// TwinCAT 3 PLC project SpeedControl
// ProgramVersion: 3.1.4020.4
// libraries:
//   Tc2_Drive, * (Beckhoff Automation GmbH)
//   Tc2_EtherCAT, * (Beckhoff Automation GmbH)
//   Tc2_MC2, * (Beckhoff Automation GmbH)
//   Tc2_Standard, * (Beckhoff Automation GmbH)
//   Tc2_System, * (Beckhoff Automation GmbH)
//   Tc2_Utilities, * (Beckhoff Automation GmbH)
//   Tc3_Module, * (Beckhoff Automation GmbH)
// project tree:
//   DUTs/ ST_COM_FTL_SpdCntrl.TcDUT, ST_COM_SpdCntrl_FTL.TcDUT, ST_COM_SpeedControl_IMD.TcDUT, ST_COM_IMD_SpdCntrl.TcDUT, ST_COM_SpeedControl_FTL.TcDUT, ST_MachPar.TcDUT, ST_OEE.TcDUT, ST_PowerMeasurement.TcDUT, ST_ProdPar.TcDUT, ST_ProductPar.TcDUT, ST_COM_SpdCntrl_IMD.TcDUT, ST_SysPar.TcDUT
//   GVLs/ GVL.TcGVL
//   / PlcTask_SpeedControl.TcTTO, RecipeManager.TcRMO (not stored)
//   POUs/SpeedControl/ FB_BlowOff.TcPOU, ST_BlowOffMachPar.TcDUT, ST_BlowOffErrors.TcDUT, ST_BlowOffProdPar.TcDUT, FB_Conveyor.TcPOU, ST_ConveyorErrors.TcDUT, ST_ConveyorMachPar.TcDUT, ST_ConveyorProdPar.TcDUT, ST_ConveyorSysPar.TcDUT
//   POUs/ HMI.TcPOU, MAIN.TcPOU, ST_Errors.TcDUT
//   Standard/ FB_Blink.TcPOU, FB_EthercatDiag.TcPOU
//   Standard/Motor/ FB_Motor.TcPOU, FB_MotorSS.TcPOU, ST_MotorErrors.TcDUT, ST_MotorSSErrors.TcDUT
//   Standard/NC_Axis/ FB_NcAxis.TcPOU, ST_NcAxis_Errors.TcDUT, ST_NcAxis_Parameters_XX.TcDUT, ST_NcAxis_SysPar.TcDUT
// (motion and I/O tree: see PLC project imd_plc)
// real-time tasks:
//   TASK PlcTask: cycle T#10ms, priority 20, ADS port 350
//   TASK PlcTask_SpeedControl: cycle T#2ms, priority 19, ADS port 351
// variable links:
//   IMD_PLC/IMD_PLC Instance <-> SpeedControl/SpeedControl Instance
//     PlcTask Inputs/MAIN.ComSC.SpeedControl_IMD <-> PlcTask_SpeedControl Outputs/MAIN.ComSpeedControl_IMD1.SpeedControl_IMD
//     PlcTask Outputs/MAIN.ComSC.IMD_SpeedControl <-> PlcTask_SpeedControl Inputs/MAIN.ComSpeedControl_IMD1.IMD_SpeedControl
//   SpeedControl/SpeedControl Instance <-> Device 2 (EtherCAT)/MCC01_2_610A1 (EK1100)/610A2 (EK1122)/Drive A-Belt / B-Spraybar (AX5201-0000-0203)
//     PlcTask_SpeedControl Inputs/MAIN.Conveyor.Belt.iDriveRef/aNetId <-> InfoData/AdsAddr/netId
//     PlcTask_SpeedControl Inputs/MAIN.Conveyor.Belt.iDriveRef/nDriveNo <-> InfoData/Chn0
//     PlcTask_SpeedControl Inputs/MAIN.Conveyor.Belt.iDriveRef/nSlaveAddr <-> InfoData/AdsAddr/port
//   SpeedControl/SpeedControl Instance <-> Device 2 (EtherCAT)/MCC01_2_610A1 (EK1100)/610A2 (EK1122)/EJBox (EP9128-0021)/EPP_SensorSpeedControl (EPP1322-0001)/Box SpeedControl (EPP6228-0022)
//     PlcTask_SpeedControl Inputs/MAIN.Conveyor.IMD1_GantryB.miSensorPitchClear <-> Module 11 (Digital Inputs)/Digital Inputs/Pin2 Ch1
//   SpeedControl/SpeedControl Instance <-> NC-Task 1 SAF/Axes/Conveyor
//     PlcTask_SpeedControl Inputs/MAIN.Conveyor.Belt.axAxis.NcToPlc <-> Outputs/ToPlc
//     PlcTask_SpeedControl Outputs/MAIN.Conveyor.Belt.axAxis.PlcToNc <-> Inputs/FromPlc

CONFIGURATION SpeedControl
    RESOURCE PLC ON TwinCAT3
        TASK PlcTask_SpeedControl(INTERVAL := T#2ms, PRIORITY := 19);
        PROGRAM MAIN WITH PlcTask_SpeedControl : MAIN;
    END_RESOURCE
END_CONFIGURATION

// ---- DUTs/ST_COM_FTL_SpdCntrl.TcDUT
TYPE ST_COM_FTL_SpdCntrl :
STRUCT
	MaximumSpeed	: LREAL; //(KO, amount of sheets/min)
	RTO				: BOOL;	//FTL is Ready to Operate state
	Stop			: BOOL;
	ES				: BOOL;
END_STRUCT
END_TYPE

// ---- DUTs/ST_COM_SpdCntrl_FTL.TcDUT
TYPE ST_COM_SpdCntrl_FTL :
STRUCT
	ReadyToRun			: BOOL;
	ES					: BOOL;
END_STRUCT
END_TYPE

// ---- DUTs/ST_COM_SpeedControl_IMD.TcDUT
TYPE ST_COM_SpeedControl_IMD :
STRUCT
	//Speedcontrol - IMD
	IMD_SpeedControl		AT %I* :ST_COM_IMD_SpdCntrl;
	SpeedControl_IMD		AT %Q* :ST_COM_SpdCntrl_IMD;
END_STRUCT
END_TYPE

// ---- DUTs/ST_COM_IMD_SpdCntrl.TcDUT
TYPE ST_COM_IMD_SpdCntrl :
STRUCT
	Stopped				: BOOL;					// IMD is in stopped state
	RTO					: BOOL;					// IMD is Ready to Operate state
	BlowOffProcessedA	: ARRAY[1..4] OF BOOL;	// signal to confirm that the blowoff has actually happend for A side
	BlowOffProcessedB	: ARRAY[1..4] OF BOOL;	// signal to confirm that the blowoff has actually happend for B side
	FormingReadyA		: BOOL;					// signal to confirm that the forming has actually started for A side
	FormingReadyB		: BOOL;					// signal to confirm that the forming has actually started for B side
	GantryA_Ready		: BOOL; 				// signal that Gantry A is in position above the conveyor and ready to blow off
	GantryB_Ready		: BOOL; 				// signal that Gantry B is in position above the conveyor and ready to blow off
	ES					: BOOL;					// Emergency stop from the IMD that also need to stop the conveyor
	MaximumSpeed		: REAL;					// theoretical maximum speed with current settings
	ActualSpeed			: REAL;					// Number of KO's in last cycle
	HMI_Reset			: BOOL;					// MZE 20190311 For testing at LoodsLanghout
END_STRUCT
END_TYPE

// ---- DUTs/ST_COM_SpeedControl_FTL.TcDUT
TYPE ST_COM_SpeedControl_FTL :
STRUCT
	//Speedcontrol - FTL
	FTL_SpeedControl		AT %I* :ST_COM_FTL_SpdCntrl;
	SpeedControl_FTL		AT %Q* :ST_COM_SpdCntrl_FTL;
END_STRUCT
END_TYPE

// ---- DUTs/ST_MachPar.TcDUT
TYPE ST_MachPar :
STRUCT
	Conveyor				: ST_ConveyorMachPar;
END_STRUCT
END_TYPE

// ---- DUTs/ST_OEE.TcDUT
TYPE ST_OEE :
STRUCT
	AmountOfSheets			 		: DINT;
	AmoundOfProductsSheets			: DINT;
	
END_STRUCT
END_TYPE

// ---- DUTs/ST_PowerMeasurement.TcDUT
TYPE ST_PowerMeasurement :
STRUCT
	ixPDOToggle		:BOOL;
	iwCurrent 		:DINT;
	iwVoltage		:DINT;
	iwActivePower	:DINT;
	iwIndex			:USINT;
	iwVariantValue	:DINT;
END_STRUCT
END_TYPE

// ---- DUTs/ST_ProdPar.TcDUT
TYPE ST_ProdPar :
STRUCT
	Conveyor			: ST_ConveyorProdPar;
	Product				: ST_ProductPar;
END_STRUCT
END_TYPE

// ---- DUTs/ST_ProductPar.TcDUT
TYPE ST_ProductPar :
STRUCT
	PlaceHolder			: BOOL;
END_STRUCT
END_TYPE

// ---- DUTs/ST_COM_SpdCntrl_IMD.TcDUT
TYPE ST_COM_SpdCntrl_IMD :
STRUCT
	StartFormingA		: BOOL;	//Speedcontrol needs the IMD to start froming for A side	
	StartFormingB		: BOOL;	//Speedcontrol needs the IMD to start froming for B side	
	StopForming			: BOOL;	//Speedcontrol needs the IMD to stop forming 
	BlowOffPulseA		: ARRAY[1..4] OF BOOL; 	//Blowoff pulses for A side
	BlowOffPulseB		: ARRAY[1..4] OF BOOL;	//Blowoff pulses for B side
	ErrSlotANotFree		: BOOL;					//Current slot for gantry A blow off was not free
	ErrSlotBNotFree		: BOOL;					//Current slot for gantry B blow off was not free	
	Modulo				: LREAL;				//Actual modulo position of the belt  
	SpeedInKo			: LREAL;				//Actual Speed that speedcontrol is dictating to the IMD
	PocketA_Blocked		: BOOL;					//Pocket is occupied and gantry is not allowed to blow off
	PocketB_Blocked		: BOOL;					//Pocket is occupied and gantry is not allowed to blow off
	ProdParameters		: ST_BlowOffProdPar;
END_STRUCT
END_TYPE

// ---- DUTs/ST_SysPar.TcDUT
TYPE ST_SysPar :
STRUCT
	Conveyor					: ST_ConveyorSysPar;
END_STRUCT
END_TYPE

// ---- POUs/SpeedControl/ST_BlowOffMachPar.TcDUT
TYPE ST_BlowOffMachPar :
STRUCT
	NrOfPitchMissedAlarm		: DINT;
END_STRUCT
END_TYPE

// ---- POUs/SpeedControl/ST_BlowOffErrors.TcDUT
TYPE ST_BlowOffErrors :
STRUCT
	PitchNotFree_Error		: BOOL;	//Designated pitch for blow off not free	
END_STRUCT
END_TYPE

// ---- POUs/SpeedControl/ST_BlowOffProdPar.TcDUT
TYPE ST_BlowOffProdPar :
STRUCT
	PitchGantry					: DINT;	//Pitch distance between sheets on gantry
	NrOfSheets					: DINT;	//Amount of sheets used on IMD
	NrOfCavities				: DINT;  // The amount of cavities (products) in one sheet.
	Modulo						: LREAL; //System parameter (5180)
	ModuloOffsetSensorFree		: REAL; //Offset on the modulo to start measuring if the pitch is free for dropping
	ModuloDetectionSensorFree	: REAL;	//How long the sensor needs to be active before alarm/skipping blow off based on modulo length
	SheetSize					: REAL;	//The width of a sheet
END_STRUCT
END_TYPE

// ---- POUs/SpeedControl/ST_ConveyorErrors.TcDUT
TYPE ST_ConveyorErrors :
STRUCT
	NCAxisError					: ST_NcAxis_Errors;
	
END_STRUCT
END_TYPE

// ---- POUs/SpeedControl/ST_ConveyorMachPar.TcDUT
TYPE ST_ConveyorMachPar :
STRUCT
	VelocityManual						: LREAL;
	VelocityAuto						: LREAL;
	InitSpeed							: LREAL;
	ModuloRamp							: DINT;	
	IMD1_Enabled						: BOOL;
	IMD2_Enabled						: BOOL;
END_STRUCT
END_TYPE

// ---- POUs/SpeedControl/ST_ConveyorProdPar.TcDUT
TYPE ST_ConveyorProdPar :
STRUCT
	BlowOff_Prod			: ST_BlowOffProdPar;
	
END_STRUCT
END_TYPE

// ---- POUs/SpeedControl/ST_ConveyorSysPar.TcDUT
TYPE ST_ConveyorSysPar :
STRUCT
	Belt					: ST_NcAxis_SysPar;
	
END_STRUCT
END_TYPE

// ---- POUs/ST_Errors.TcDUT
TYPE ST_Errors :
STRUCT
	exEmergency						: ARRAY[1..GVL.MAX_ZONES+1] OF BOOL;  (*Emergecy Stop Active, Index=Zone, 1=Stacker, 2=Zipper, 3=Bundle Buffer track, 4=Vertical denester, 5=Bundle Outfeed // stop buttons.*)
	exEmStop						: BOOL;
	
	ex24VoltError1					: BOOL; 
	ex24VoltError2					: BOOL;
	
	exUpsAlarm						: BOOL;
	
	exAtteptedStartWithNoProduct	: BOOL;
	
	ConveyorErrors 					: ST_ConveyorErrors;
	
	
END_STRUCT
END_TYPE

// ---- Standard/Motor/ST_MotorErrors.TcDUT
TYPE ST_MotorErrors :
STRUCT	
	Thermal					: BOOL;
	Maintenance				: BOOL;
END_STRUCT
END_TYPE

// ---- Standard/Motor/ST_MotorSSErrors.TcDUT
TYPE ST_MotorSSErrors :
STRUCT	
	SofstarterFailure		: BOOL;
	Maintenance				: BOOL;
END_STRUCT
END_TYPE

// ---- Standard/NC_Axis/ST_NcAxis_Errors.TcDUT
TYPE ST_NcAxis_Errors :
STRUCT
	exDriveStatus: BOOL;
	///~ (OPC:1:available for OPC Clients) 
	exDrivePower: BOOL;
	///~ (OPC:1:available for OPC Clients) 
	exDriveJog: BOOL;
	///~ (OPC:1:available for OPC Clients) 
	exDriveReset: BOOL;
	///~ (OPC:1:available for OPC Clients) 

	exDriveAbsoluut				: BOOL;
	exDriveVelocity				: BOOL;
	exDriveStop					: BOOL;
	exWriteParameter			: BOOL;
	exReadParameter				: BOOL;
	exHome						: BOOL;
	exLagError					: BOOL;	(*Lag error*)
	
END_STRUCT
END_TYPE

// ---- Standard/NC_Axis/ST_NcAxis_Parameters_XX.TcDUT
TYPE ST_NcAxis_Parameters_XX :
STRUCT
	VelocityAuto		:	LREAL;	(*Automatic speed*)
	VelocityManual		:	LREAL; 	(*manual speed*)
	VelocityInit		:	LREAL;	(*init speed*)
	HomePosition		:	LREAL;	(*Homing position*)
	Acceleration		:	LREAL;  (*Acceleration speed*)
	Deceleration		:	LREAL;  (*Deceleration speed*)
	DecelerationStop	:	LREAL:=1000;	(*Deceleration *)	

END_STRUCT
END_TYPE

// ---- Standard/NC_Axis/ST_NcAxis_SysPar.TcDUT
TYPE ST_NcAxis_SysPar :
STRUCT
	PositionBias			: LREAL;(* From absolute encoder *)
	IDXGRP				:UDINT := 16#5011;

END_STRUCT
END_TYPE

// ---- GVLs/GVL.TcGVL

VAR_GLOBAL PERSISTENT
	PersMachPar					: ST_MachPar;
	PersSysPar					: ST_SysPar;
END_VAR
VAR_GLOBAL CONSTANT
	MAX_ZONES					: INT:= 7;
END_VAR

// ---- POUs/MAIN.TcPOU
PROGRAM MAIN
VAR
	mxReset									: BOOL;
	mxEmergency								: BOOL;
	mxAutoMode								: BOOL; (* "1" = Auto, "0" = Manual *)
	mxFirstCycle							: BOOL;
	
	Conveyor								: FB_Conveyor;
	Blink									: FB_Blink;
	
	mxHMI_Start								: BOOL;
	mxHMI_Stop								: BOOL;
	mxHMI_Pause								: BOOL;
	mxHMI_Reset								: BOOL;
	//mxHMI_StartInit							: BOOL;
	//mxHMI_StopInit							: BOOL;
	mxProductLoaded							: BOOL;
	mxMachineInRest							: BOOL;
	
	mxHMI_StartState						: BOOL;
	mxHMI_StopState							: BOOL;
	mxHMI_PauseState						: BOOL;
	
	RT_Start								: R_TRIG;
	RT_Stop									: R_TRIG;
	RT_Pause								: R_TRIG;
	RT_StartInit							: R_TRIG;
	RT_StopInit								: R_TRIG;
	
	qxLightGreen							AT %Q* : BOOL;
	qxLightYellow							AT %Q* : BOOL;
	qxLightRed								AT %Q* : BOOL;
	qxAlarmHorn								AT %Q* : BOOL;

	(*Added by bateu*)
	ix24VoltError1							AT %I* : BOOL;
	ix24VoltError2							AT %I* : BOOL;
	
	L1										AT %I* : ST_PowerMeasurement;
	L2										AT %I* : ST_PowerMeasurement;
	L3										AT %I* : ST_PowerMeasurement;		
	
	Errors									: ST_Errors;
	
(*TwinSAFE*)
	ixTwinSafe_SafetyRelay 					AT %I*:ARRAY[1..GVL.MAX_ZONES] OF BOOL; (* couple to zones in Safety programm FB outputs *)
	qxTwinSafe_Reset						AT %Q*: BOOL;

	FbError 								AT %I*: BOOL;
	ComErr 									AT %I*: BOOL;
	OutErr 									AT %I*: BOOL;
	
	(* Em Stops *)
	SR_exEmergency							: ARRAY[1..GVL.MAX_ZONES] OF SR; (* Emergency of the zones *)
	SR_EmStop								: SR;
	
	(*24V error*)
	SR_24VError1							: SR;
	SR_24VError2							: SR;
	
	SR_AttemptedStartWithNoProductLoaded	: SR;

	T_HMIReset								: TON;
	
	MachPar									: ST_MachPar;
	ProdPar									: ST_ProdPar;	
	SysPar									: ST_SysPar;
	(* Persistent vars*)
	ChkMachPar								: ST_MachPar;
	CmpMachPar								: DINT;
	ChkSysPar								: ST_SysPar;
	CmpSysPar								: DINT;
	RTRIG_WritePersistent					: R_TRIG;
	FB_WritePersistentData					: WritePersistentData;
	FB_GetCurTaskIdx						: GETCURTASKINDEX;
	T_WritePersistent						: TON;
	mxErrorInit								: BOOL;
	FT_AutoMode								: F_Trig;
	RT_MasterReset							: R_trig;
	mxInitialized							: BOOL;
	iwDevID									AT %I* :UINT;
	iAmsNetID								AT %I* :ARRAY [0..5] OF BYTE;
	iwSlaveCount							AT %I* :UINT;
	iwCfgSlaveCount							AT %I* :UINT;
	iwDevState								AT %I* :UINT;
	EtherCatDiag							: FB_EtherCATDiag;
	AmsNetID								: STRING;
	DeviceID								: INT;

	mxHMI_Stopping							: BOOL;
	
	Phase1									: REAL;
	Phase2									: REAL;
	Phase3									: REAL;

	
	ixMainSwitchOFF							AT %I* : BOOL;	
	ixUPS_Alarm								AT %I* : BOOL;
	ixUPS_BatMode							AT %I* : BOOL;
	ixUPS_Charge							AT %I* : BOOL;
	
	qxPcRemoteOff							AT %Q* : BOOL;
	
	PlcCycleTime     						: REAL := 10.0;
	RT_PauseReq								: R_TRIG;
	
	EmButtons								: BOOL;
	
	T_BatteryMode							: TON;
	T_MaintSwitch							: TON;
	SR_UPSAlarm								: SR;
	
	ComSpeedControl_IMD1					: ST_COM_SpeedControl_IMD;
	ComSpeedControl_IMD2					: ST_COM_SpeedControl_IMD;
	ComSpeedControl_FTL						: ST_COM_SpeedControl_FTL;
	
	RT_StopByFTL							: R_TRIG;
	mxStopByFTL								: BOOL;
	RT_StartByFTL							: R_TRIG;
END_VAR

// 					Object Calls				//
FB_GetCurTaskIdx();
mxFirstCycle:= _TaskInfo[FB_GetCurTaskIdx.index].FirstCycle;
PlcCycleTime:= UDINT_TO_REAL(_TaskInfo[FB_GetCurTaskIdx.index].CycleTime/10000);
RemanentData();
Blink();
Error();
Objects();
HMI();
OEEE();
COM_IMD();

// 					R_Trigs.					//
RT_Start(CLK:= mxHMI_Start);
RT_Stop(CLK:= mxHMI_Stop OR Conveyor.mxErrorStopInPos); 
RT_StartByFTL(CLK:= ComSpeedControl_FTL.FTL_SpeedControl.RTO);
RT_StopByFTL(CLK:=NOT ComSpeedControl_FTL.FTL_SpeedControl.RTO);
RT_Pause(CLK:= mxHMI_Pause);
//RT_StartInit(CLK:= mxHMI_StartInit);
//RT_StopInit(CLK:= mxHMI_StopInit);
RT_MasterReset(CLK:= NOT mxAutoMode);
//RT_PauseReq(ClK:=Conveyor.mxErrorStopInPos);
//mxInitialized:= InMoldDrying.mxInitialized AND ProductHandling.mxInitialized;
mxMachineInRest := NOT Conveyor.mxCycleBusy;


// 					Start machine				//
IF (RT_Start.Q OR (mxStopByFTL AND RT_StartByFTL.Q)) AND mxAutoMode AND NOT Conveyor.mxErrorStopInPos THEN  
	Conveyor.M_StartCycle(); 
	mxHMI_Stopping :=FALSE;
	mxStopByFTL := FALSE;
END_IF

//					Normal stop					//
IF (RT_Stop.Q OR RT_StopByFTL.Q) AND mxAutoMode THEN  
	Conveyor.M_StopCycle();  
	mxHMI_Stopping := TRUE;	
	mxStopByFTL := FALSE;	
	IF RT_StopByFTL.Q AND Conveyor.mxCycleBusy THEN
		mxStopByFTL := TRUE;	
	END_IF
END_IF

//					Stop direct error			//
IF mxErrorInit OR Conveyor.mxErrorInit (*OR ComSpeedControl_IMD1.IMD_SpeedControl.ES OR ComSpeedControl_IMD2.IMD_SpeedControl.ES*) THEN
	Conveyor.M_StopDirect();
	mxStopByFTL := FALSE;
END_IF

//					HMI stop button color		//
IF mxHMI_Stopping THEN
	mxHMI_StopState := TRUE;
ELSIF NOT Conveyor.mxCycleBusy THEN
	mxHMI_StopState := TRUE;
	mxHMI_Stopping := FALSE;
ELSE
	mxHMI_StopState := FALSE;
	mxHMI_Stopping := FALSE;	
END_IF

(*
//					Signal light				//
qxLightEmStopImdFront:= qxLightEmStopImdBack:= qxLightEmStopGantryA_Front:= qxLightEmStopGantryA_Back:= qxLightEmStopGantryB_Front:= qxLightEmStopGantryB_Back := 
	Errors.exEmergency[1] OR Errors.exEmergency[2] OR Errors.exEmergency[3] OR Errors.exEmergency[4] OR Errors.exEmergency[5] OR Errors.exEmergency[6] OR Errors.exEmergency[7];
qxLightRed:= HMI.mxError;
qxLightGreen:= mxHMI_StartState := (InMoldDrying.mxCycleBusy OR ProductHandling.mxCycleBusy) AND NOT mxHMI_PauseState;
qxLightYellow:= FALSE;
*)
mxHMI_StartState := Conveyor.mxCycleBusy;

//					Reseting					//
T_HMIReset(IN:= mxHMI_Reset,PT:=T#1S);
IF T_hmiReset.Q THEN mxHMI_Reset:=FALSE; END_IF

mxReset:= qxTwinSafe_Reset:= mxHMI_Reset;

//					Master reset				//
IF RT_MasterReset.Q THEN
	Conveyor.mxResetCycleState := TRUE;
	mxStopByFTL := FALSE;
END_IF

// Get AMS net id and device id for ethercat topology
AmsNetID:= F_CreateAmsNetId(iAmsNetID);
DeviceID:= UINT_TO_INT(iwDevID);

mxHMI_Start := FALSE;
mxHMI_Stop := FALSE;
mxHMI_Pause := FALSE;

// Shut of PC when on battery mode or when power was switched off:
//T_BatteryMode(IN:=ixUPS_BatMode, PT:=T#30S);
//T_MaintSwitch(IN:=NOT ixMainSwitchOFF);

// Uncomment when timers are tested.
//qxPcRemoteOff := T_BatteryMode.Q OR T_MaintSwitch.Q;

ACTION COM_IMD:
ComSpeedControl_IMD1.SpeedControl_IMD.ProdParameters :=  ProdPar.Conveyor.BlowOff_Prod;
ComSpeedControl_IMD2.SpeedControl_IMD.ProdParameters :=  ProdPar.Conveyor.BlowOff_Prod;
mxHMI_Reset := ComSpeedControl_IMD1.IMD_SpeedControl.HMI_Reset;
END_ACTION

ACTION Error:
(*Emergency Stop Active Zone x,  Index=Zone , 1=Takeout/Gantr A, 2=Imd Left, 3=Imd Middle, 4=Imd Right, 5=Takeout/Gantry B*, 6=Gantry B *)
(*SR_exEmergency[1](SET1:= NOT ixTwinSafe_SafetyRelay[1], RESET:=ixTwinSafe_SafetyRelay[1] , Q1=>Errors.exEmergency[1] );
SR_exEmergency[2](SET1:= NOT ixTwinSafe_SafetyRelay[2], RESET:=ixTwinSafe_SafetyRelay[2] , Q1=>Errors.exEmergency[2] );
SR_exEmergency[3](SET1:= NOT ixTwinSafe_SafetyRelay[3], RESET:=ixTwinSafe_SafetyRelay[3] , Q1=>Errors.exEmergency[3] );
SR_exEmergency[4](SET1:= NOT ixTwinSafe_SafetyRelay[4], RESET:=ixTwinSafe_SafetyRelay[4] , Q1=>Errors.exEmergency[4] );
SR_exEmergency[5](SET1:= NOT ixTwinSafe_SafetyRelay[5] , RESET:=ixTwinSafe_SafetyRelay[5], Q1=>Errors.exEmergency[5] );
SR_exEmergency[6](SET1:= NOT ixTwinSafe_SafetyRelay[6] , RESET:=ixTwinSafe_SafetyRelay[6], Q1=>Errors.exEmergency[6] );
SR_exEmergency[7](SET1:= NOT ixTwinSafe_SafetyRelay[7] , RESET:=ixTwinSafe_SafetyRelay[7], Q1=>Errors.exEmergency[7] );

(*24V error*)
SR_24VError1(Set1:=NOT ix24VoltError1, Reset:=mxReset, Q1=>Errors.ex24VoltError1); 
SR_24VError2(Set1:=NOT ix24VoltError2, Reset:=mxReset, Q1=>Errors.ex24VoltError2); 
SR_UPSAlarm(Set1:=NOT ixUPS_Alarm, Reset:=mxReset, Q1=>Errors.exUpsAlarm);

SR_AttemptedStartWithNoProductLoaded(Set1:=NOT mxProductLoaded AND (RT_Start.Q OR RT_StartInit.Q), Reset:=mxReset, Q1=>Errors.exAtteptedStartWithNoProduct);

EtherCatDiag(
	SlaveCount:=	iwSlaveCount,
	CfgSlaveCount:=	iwCfgSlaveCount,
	DevState:=		iwDevState);

Errors.exEmergency[8]	:=EmButtons := Errors.exEmStop;
	
mxEmergency := Errors.exEmergency[1] OR Errors.exEmergency[2] OR Errors.exEmergency[3] OR 
Errors.exEmergency[4] OR Errors.exEmergency[5] OR Errors.exEmergency[6] OR Errors.exEmergency[7] OR EmButtons;

mxErrorInit:= EmButtons;*)
END_ACTION

ACTION Objects:
Conveyor(
	mxReset:= mxReset, 
	mxEmergency:=  FALSE, (*ComSpeedControl_IMD1.IMD_SpeedControl.ES OR ComSpeedControl_IMD2.IMD_SpeedControl.ES,*)
	mxAutoMode:= mxAutoMode,
	mxFirstCycle:= mxFirstCycle,
	MachParameters 	:= MachPar.Conveyor,
	ProdParameters 	:= ProdPar.Conveyor,
	SysParameters	:= SysPar.Conveyor,
	IMD1_COM_IN		:= ComSpeedControl_IMD1.IMD_SpeedControl,
	IMD1_COM_OUT	:= ComSpeedControl_IMD1.SpeedControl_IMD,
	IMD2_COM_IN		:= ComSpeedControl_IMD2.IMD_SpeedControl,
	IMD2_COM_OUT	:= ComSpeedControl_IMD2.SpeedControl_IMD,
	FTL_COM_IN		:= ComSpeedControl_FTL.FTL_SpeedControl,
	FTL_COM_OUT		:= ComSpeedControl_FTL.SpeedControl_FTL,
);
END_ACTION

ACTION OEEE:

// Calculate the voltage to normal format (000.00V)
Phase1 := DINT_TO_REAL(L1.iwVoltage) / 10000.0;
Phase2 := DINT_TO_REAL(L2.iwVoltage) / 10000.0;
Phase3 := DINT_TO_REAL(L3.iwVoltage) / 10000.0;
END_ACTION

ACTION RemanentData:
IF mxFirstCycle THEN
	MachPar:= PersMachPar;
	SysPar:= PersSysPar;
END_IF

CmpMachPar:= MEMCMP(ADR(MachPar), ADR(ChkMachPar),SIZEOF(ChkMachPar));
CmpSysPar:= MEMCMP(ADR(SysPar), ADR(ChkSysPar),SIZEOF(ChkSysPar));

(* Backup every x min. the persistent parameters *)
T_WritePersistent(IN:= NOT T_WritePersistent.Q , PT:=T#5M);

RTrig_WritePersistent(CLK:= (CmpMachPar <> 0) OR (CmpSysPar <> 0));

IF RTRIG_WritePersistent.Q THEN
	PersMachPar:= MachPar;
	PersSysPar:= SysPar;
	FB_WritePersistentData(NETID:='', PORT:=852, START:=TRUE, TMOUT:=T#1S );	
ELSE
	FB_WritePersistentData(NETID:='', PORT:=852, START:=FALSE, TMOUT:=T#1S );
END_IF

ChkMachPar:= MachPar;
ChkSysPar:= SysPar;
END_ACTION

END_PROGRAM

// ---- POUs/SpeedControl/FB_Conveyor.TcPOU
FUNCTION_BLOCK FB_Conveyor
VAR CONSTANT
	sCycleStateTextDef: ARRAY[0..10]  OF STRING :=	
		['State 0: Wait for Start',
		'State 1: Start conveyor',
		'State 2: Start Gantries',
		'State 3: Spare',
		'State 4: Spare',
		'State 5: Spare',
		'State 6: Belt running, control speed','7','8','9',
		'State 10: Error'];
	
	tCycleStateTimeouts: ARRAY[0..10] OF TIME := 
		[T#10S,T#10S,T#60S,T#10S,T#10S,T#10S,T#10S,T#10S,T#10S,T#10S,
		T#10S];

END_VAR
VAR_INPUT
	mxResetCycleState				: BOOL;
	mxReset							: BOOL;	(*Reset Error*)
	mxEmergency						: BOOL;
	mxAutoMode						: BOOL; (* TRUE = Automode *)
	mxFirstCycle					: BOOL;

END_VAR
VAR_IN_OUT
	MachParameters					: ST_ConveyorMachPar;
	ProdParameters					: ST_ConveyorProdPar;
	SysParameters					: ST_ConveyorSysPar;
	
	IMD1_COM_IN						: ST_COM_IMD_SpdCntrl;
	IMD1_COM_OUT					: ST_COM_SpdCntrl_IMD;
	IMD2_COM_IN						: ST_COM_IMD_SpdCntrl;
	IMD2_COM_OUT					: ST_COM_SpdCntrl_IMD;
	
	FTL_COM_IN						: ST_COM_FTL_SpdCntrl;
	FTL_COM_OUT						: ST_COM_SpdCntrl_FTL;
END_VAR
VAR_OUTPUT
	(*Errors*)
	Errors							: ST_ConveyorErrors;
	mxErrorInit						: BOOL;
	mxErrorStopinPos				: BOOL;		(* Error, stop in position. Only reset neccesary *)

(* State vars *)
	mxCycleBusy						: BOOL;
	
(* Vars *)	
	mrActModPos						: LREAL;
END_VAR
VAR
(* State vars *)
	miCycleState					: INT :=0;
	miCycleOldstate					: INT :=0;
	mxCycleTransitionState			: BOOL := FALSE;
	sCycleStateText					: STRING;
	exCycleTimeOut					: BOOL;		(* Timeout for the whole programcycle *)
	CycleTimeout					: TON;
	CycleTimeOutUpFlank				: R_TRIG;
	mxCycleTimeoutEnable			: BOOL;
	CycleTime						: REAL;
	mxCycleHasError					: BOOL;
	miStopState						: INT;
	mxStartCycle					: BOOL;
	mxStopCycle						: BOOL;
	mxStopDirect					: BOOL;
	
	(* Objects *)
	Belt							: FB_NcAxis;
	IMD1_GantryA					: FB_BlowOff;
	IMD1_GantryB					: FB_BlowOff;
	IMD2_GantryA					: FB_BlowOff;
	IMD2_GantryB					: FB_BlowOff;

	mrSetpointPosition				: LREAL;
	mrActPosBeltSaved				: LREAL;	
	
	(* Internal calculating values *)
	mrModuloStart_offset			: LREAL;
	mdModuloCount					: DINT;
	RT_ModuloCount					: R_TRIG;
	mrCalculateSpeedIMD1			: LREAL;
	mrCalculateSpeedIMD2			: LREAL;
	mrAllowdKObyFTL					: LREAL;
	mrCalculateSpeedFTL				: LREAL;
	StartSpeedConveyorAuto			: LREAL;	
	mrSetRunSpeed					: LREAL;	
	miNrOfIMD						: INT := 2; //Always calculate based on two IMD enabled
	mrSetRunSpeedOld				: LREAL;
	T_Stopping						: TON;
END_VAR

mrActModPos:= Belt.axAxis.NcToPlc.ModuloActPos;

Error();
Cycle();
Objects();

ACTION Cycle:
(*StateChange (Transition)  Signalgeneration*)
mxCycleTransitionState:=(miCycleState<>miCycleOldstate);
(*State text*)
sCycleStateText:=sCycleStateTextDef[miCycleState];
(*Timeout Watchdog for Statemachine*)
mxCycleTimeoutEnable:=NOT (miCycleState=0 OR miCycleState=6) AND NOT mxReset;

CycleTimeout(IN:=mxCycleTimeoutEnable, PT:=tCycleStateTimeouts[miCycleState] );
CycleTimeOutUpFlank(CLK:=CycleTimeout.Q );
miCycleOldstate:=miCycleState;

(*Set Errorbit when Raising edge of Timeout has been detected*)
IF CycleTimeOutUpFlank.Q THEN
	exCycleTimeOut:=TRUE; 			(* 1 Timeout for the whole programcycle *)
END_IF

(*Function to reset the Statemachine*)
IF mxResetCycleState THEN
	mxResetCycleState:= FALSE;
	miCycleState:=0;
	miCycleOldstate:=miCycleState;
	mxCycleTransitionState:=FALSE;
	mdModuloCount := 0;
	
	IMD1_GantryA.mxResetCycleState := TRUE;
	IMD1_GantryB.mxResetCycleState := TRUE;
	IMD2_GantryA.mxResetCycleState := TRUE;
	IMD2_GantryB.mxResetCycleState := TRUE;
	
	T_Stopping.IN := FALSE;
	IMD1_COM_OUT.StopForming := FALSE;
    IMD2_COM_OUT.StopForming := FALSE;
		
	mxStartCycle:= FALSE;
	mxStopCycle:= FALSE;
	mxStopDirect:= FALSE;
	Belt.M_Stop();
END_IF

(*Definition State has Error*)
mxCycleHasError:=FALSE;

(*Calculate modulo offset positions gantry*)
	IF ProdParameters.BlowOff_Prod.Modulo = 0 THEN
		ProdParameters.BlowOff_Prod.Modulo := 4620;
	END_IF
	IMD1_GantryA.mrModuloOffset:= (ProdParameters.BlowOff_Prod.Modulo/4)*1;
	IMD1_GantryB.mrModuloOffset:= (ProdParameters.BlowOff_Prod.Modulo/4)*3;
	IMD2_GantryA.mrModuloOffset:= 0;
	IMD2_GantryB.mrModuloOffset:= (ProdParameters.BlowOff_Prod.Modulo/4)*2;

(*Calculate allowed speeds from Communication partners *)
	(*IF MachParameters.IMD1_Enabled AND MachParameters.IMD2_Enabled THEN		//For now speed of the conveyor will always be based on 2 IMD's
		miNrOfIMD := 2;
	ELSIF MachParameters.IMD1_Enabled OR MachParameters.IMD2_Enabled THEN
		miNrOfIMD := 1;	
	END_IF*)
	
	IF ProdParameters.BlowOff_Prod.NrOfSheets = 0 THEN
		ProdParameters.BlowOff_Prod.NrOfSheets := 3;
	END_IF
	
	IF ((IMD1_COM_IN.MaximumSpeed = 0) AND IMD1_COM_IN.RTO) THEN
		mrCalculateSpeedIMD1 := StartSpeedConveyorAuto;
	ELSE
		mrCalculateSpeedIMD1 := ((IMD1_COM_IN.MaximumSpeed-0.05) * miNrOfIMD)*((ProdParameters.BlowOff_Prod.Modulo/4)/60);
	END_IF
	IF ((IMD2_COM_IN.MaximumSpeed = 0) AND IMD2_COM_IN.RTO) THEN
		mrCalculateSpeedIMD2 := StartSpeedConveyorAuto;
	ELSE
		mrCalculateSpeedIMD2 := ((IMD2_COM_IN.MaximumSpeed-0.05) * miNrOfIMD)*((ProdParameters.BlowOff_Prod.Modulo/4)/60);	
	END_IF
	mrAllowdKObyFTL := (FTL_COM_IN.MaximumSpeed/ProdParameters.BlowOff_Prod.NrOfSheets)/miNrOfIMD; 	
	mrCalculateSpeedFTL := (mrAllowdKObyFTL * miNrOfIMD)*((ProdParameters.BlowOff_Prod.Modulo/4)/60);
	StartSpeedConveyorAuto := (MachParameters.VelocityAuto * miNrOfIMD)*((ProdParameters.BlowOff_Prod.Modulo/4)/60);
	IF StartSpeedConveyorAuto > mrCalculateSpeedFTL THEN
		StartSpeedConveyorAuto := mrCalculateSpeedFTL;
	END_IF
	
	IF (MachParameters.IMD1_Enabled AND IMD1_COM_IN.RTO) AND (MachParameters.IMD2_Enabled AND IMD2_COM_IN.RTO) THEN
		IF ( mrCalculateSpeedIMD1 <= mrCalculateSpeedFTL ) AND (mrCalculateSpeedIMD2 <= mrCalculateSpeedFTL) THEN
			IF (mrCalculateSpeedIMD1 <= mrCalculateSpeedIMD2) THEN
				mrSetRunSpeed := mrCalculateSpeedIMD1;
			ELSE
				mrSetRunSpeed := mrCalculateSpeedIMD2;
			END_IF
		ELSIF ( mrCalculateSpeedIMD1 <= mrCalculateSpeedFTL ) AND (mrCalculateSpeedIMD2 >= mrCalculateSpeedFTL) THEN
			mrSetRunSpeed := mrCalculateSpeedIMD1;
		ELSIF ( mrCalculateSpeedIMD1 >= mrCalculateSpeedFTL ) AND (mrCalculateSpeedIMD2 <= mrCalculateSpeedFTL) THEN
			mrSetRunSpeed := mrCalculateSpeedIMD2;
		ELSE
			mrSetRunSpeed := mrCalculateSpeedFTL;
		END_IF	
	ELSIF MachParameters.IMD1_Enabled AND IMD1_COM_IN.RTO THEN
		IF mrCalculateSpeedIMD1 <= mrCalculateSpeedFTL THEN
			mrSetRunSpeed := mrCalculateSpeedIMD1;
		ELSE
			mrSetRunSpeed := mrCalculateSpeedFTL;
		END_IF
	ELSIF MachParameters.IMD2_Enabled AND IMD2_COM_IN.RTO THEN
		IF mrCalculateSpeedIMD2 <= mrCalculateSpeedFTL THEN
			mrSetRunSpeed := mrCalculateSpeedIMD2;
		ELSE
			mrSetRunSpeed := mrCalculateSpeedFTL;
		END_IF
	ELSIF NOT IMD1_COM_IN.RTO AND NOT IMD2_COM_IN.RTO THEN
		mrSetRunSpeed := StartSpeedConveyorAuto;	
	END_IF
	IF mrSetRunSpeed < StartSpeedConveyorAuto AND (( MachParameters.IMD1_Enabled AND IMD1_COM_IN.RTO) OR (MachParameters.IMD2_Enabled AND IMD2_COM_IN.RTO)) THEN
			mrSetRunSpeed := StartSpeedConveyorAuto;
	END_IF
	
(*Time delay speed control stopped to IMD's*)
	T_Stopping(PT:=T#5S);
	IF T_Stopping.Q THEN
		IMD1_COM_OUT.StopForming := TRUE;
        IMD2_COM_OUT.StopForming := TRUE;
	END_IF
	
(*Cycle State's*)
CASE miCycleState OF
	0:
	(*
		- wait for startcycle
		- Move belt with velo
  
	*)
		IF mxStartCycle THEN
			mxStartCycle:= FALSE;
			T_Stopping.IN := FALSE;
			IMD1_COM_OUT.StopForming := FALSE;
            IMD2_COM_OUT.StopForming := FALSE;
			
			miCycleState:= 1;
		END_IF	

	(* Move belt *)
	1:
		IF mxStopDirect THEN
			mxStopDirect:= FALSE;
			
			miCycleState:= 25;
		ELSIF mxStopCycle THEN
			mxStopCycle:= FALSE;

			mrActPosBeltSaved:= Belt.ActPosition;		
	
			miStopState:= miCycleState;
			miCycleState:= 20;
		ELSIF FTL_COM_IN.RTO THEN
			mdModuloCount := 0;
			IF StartSpeedConveyorAuto > mrCalculateSpeedFTL THEN
				mrSetRunSpeed := mrCalculateSpeedFTL;
			ELSE
				mrSetRunSpeed := StartSpeedConveyorAuto;
			END_IF
			Belt.M_MoveVelocity(Velocity:= mrSetRunSpeed, Direction:= MC_Positive_Direction);
	
			miCycleState := 2;
				
		END_IF
		
	(* Start first Gantry *)	
	2:	
		IF mxStopDirect THEN
			mxStopDirect:= FALSE;
			
			miCycleState:= 25;
		ELSIF mxStopCycle THEN
			mxStopCycle:= FALSE;

			mrActPosBeltSaved:= Belt.ActPosition;		
	
			miStopState:= miCycleState;
			miCycleState:= 20;
		ELSE
		
			IF mrActModPos >= (IMD2_GantryA.mrModuloOffset - mrModuloStart_offset) AND  mrActModPos <= (IMD2_GantryA.mrModuloOffset + mrModuloStart_offset) THEN
				IMD2_GantryA.M_StartCycle();
			ELSIF mrActModPos >= (IMD1_GantryA.mrModuloOffset - mrModuloStart_offset) AND  mrActModPos <= (IMD1_GantryA.mrModuloOffset + mrModuloStart_offset) THEN
				IMD1_GantryA.M_StartCycle();
			ELSIF mrActModPos >= (IMD2_GantryB.mrModuloOffset - mrModuloStart_offset) AND  mrActModPos <= (IMD2_GantryB.mrModuloOffset + mrModuloStart_offset) THEN
				IMD2_GantryB.M_StartCycle();		
			ELSIF mrActModPos >= (IMD1_GantryB.mrModuloOffset - mrModuloStart_offset) AND  mrActModPos <= (IMD1_GantryB.mrModuloOffset + mrModuloStart_offset) THEN
				IMD1_GantryB.M_StartCycle();			
			END_IF
			
			IF IMD1_GantryA.mxCycleBusy AND IMD1_GantryB.mxCycleBusy AND IMD2_GantryA.mxCycleBusy AND IMD2_GantryB.mxCycleBusy THEN
				miCycleState:= 6;
			END_IF

		END_IF
	
		
	(* Speed control *)	
	6:
		IF mxStopDirect THEN
			mxStopDirect:= FALSE;
			
			miCycleState:= 25;
		ELSIF mxStopCycle THEN
			mxStopCycle:= FALSE;

			mrActPosBeltSaved:= Belt.ActPosition;		
	
			miStopState:= miCycleState;
			miCycleState:= 20;
		ELSE
			RT_ModuloCount(CLK:= mrActModPos >= (ProdParameters.BlowOff_Prod.Modulo - ProdParameters.BlowOff_Prod.PitchGantry));
			IF 	RT_ModuloCount.Q THEN
				mdModuloCount := mdModuloCount + 1;
			END_IF
			(*IF (Belt.ActVelocity < mrSetRunSpeed) AND (mrSetRunSpeed > 0) THEN
				Belt.M_MoveVelocity(Velocity:= mrSetRunSpeed, Direction:= MC_Positive_Direction);
			END_IF*)
			IF (mdModuloCount >=  MachParameters.ModuloRamp) OR (mrSetRunSpeed = mrCalculateSpeedFTL) OR (mrSetRunSpeed < mrSetRunSpeedOld) THEN
				mdModuloCount := 0;
				Belt.M_MoveVelocity(Velocity:= mrSetRunSpeed, Direction:= MC_Positive_Direction);
			END_IF			
		END_IF	
		
	
	(* Stop Cycle, stop belt after x mm*)
	20:
		IF mxStopDirect THEN
			mxStopDirect:= FALSE;
			
			miCycleState:= 25;
		ELSE 
			mxStopCycle:= FALSE;
			mdModuloCount := 0;
			
			Belt.M_Stop();	
			IMD1_GantryA.M_StopCycle();
			IMD1_GantryB.M_StopCycle();
			IMD2_GantryA.M_StopCycle();
			IMD2_GantryB.M_StopCycle();
			T_Stopping.IN := TRUE;
			//IMD1_COM_OUT.StopForming := TRUE;
			//IMD2_COM_OUT.StopForming := TRUE;
			
			IF NOT Belt.axStatus.Moving OR Belt.axStatus.StandStill THEN		
				miCycleState:= 21;
			END_IF
		END_IF

	21:
		IF mxStopDirect THEN
			mxStopDirect:= FALSE;
			
			miCycleState:= 25;
		ELSIF mxStartCycle THEN		
			T_Stopping.IN := FALSE;	
			mxStartCycle := FALSE;
			
			miCycleState:= 22;			
		END_IF
	
	(* wait for FTL *)	
	22:
		IF mxStopDirect THEN
			mxStopDirect:= FALSE;
			
			miCycleState:= 25;
		ELSIF FTL_COM_IN.RTO THEN		

			IMD1_GantryA.M_StartCycle();
			IMD1_GantryB.M_StartCycle();
			IMD2_GantryA.M_StartCycle();
			IMD2_GantryB.M_StartCycle();
			
			IMD1_COM_OUT.StopForming := FALSE;
			IMD2_COM_OUT.StopForming := FALSE;
			
			IF StartSpeedConveyorAuto > mrCalculateSpeedFTL THEN
				mrSetRunSpeed := mrCalculateSpeedFTL;
			ELSE
				mrSetRunSpeed := StartSpeedConveyorAuto;
			END_IF
			Belt.M_MoveVelocity(Velocity:= mrSetRunSpeed, Direction:= MC_Positive_Direction);
			
			miCycleState:= miStopState;			
		END_IF

	(* Stop Direct *)
	25:			
		mxStartCycle:= FALSE;
		mxStopCycle:= FALSE;
		mxStopDirect:= FALSE;
		mdModuloCount := 0;
		
		IMD1_GantryA.M_StopDirect();
		IMD1_GantryB.M_StopDirect();
		IMD2_GantryA.M_StopDirect();
		IMD2_GantryB.M_StopDirect();
		
		T_Stopping.IN := TRUE;
		//IMD1_COM_OUT.StopForming := TRUE;
		//IMD2_COM_OUT.StopForming := TRUE;
		
		Belt.M_Stop();

		miCycleState:= 0;
END_CASE

mxCycleBusy:= miCycleState<>0 AND miCycleState <>21;
IMD1_COM_OUT.Modulo := IMD2_COM_OUT.Modulo := mrActModPos;
IMD1_COM_OUT.SpeedInKo := IMD2_COM_OUT.SpeedInKo := (mrSetRunSpeed/((ProdParameters.BlowOff_Prod.Modulo/4)/60))/miNrOfIMD;
mrSetRunSpeedOld := mrSetRunSpeed;
END_ACTION

ACTION Error:


(*************************************************************************************************)
mxErrorStopinPos:= Belt.ErrorStop;
END_ACTION

METHOD M_StartCycle

IF NOT mxCycleBusy THEN
	mxStartCycle:= TRUE;	
END_IF
END_METHOD

METHOD M_StopCycle

IF mxCycleBusy THEN 
	mxStopCycle:= TRUE; 
END_IF
END_METHOD

METHOD M_StopDirect

IF mxCycleBusy THEN
	mxStopDirect:= TRUE;	
END_IF
END_METHOD

ACTION Objects:
IMD1_GantryA(
	mxReset							:= mxReset,
	mxEmergency						:= mxEmergency,
	mxAutoMode						:= mxAutoMode,
	mrActModulo						:= mrActModPos,
	ProdPar							:= ProdParameters.BlowOff_Prod,
	COM_IMD_Stopped					:= IMD1_COM_IN.Stopped,
	COM_IMD_RTO						:= IMD1_COM_IN.RTO,
	COM_StartFormingReady			:= IMD1_COM_IN.FormingReadyA,
	COM_BlownOffProcessed			:= IMD1_COM_IN.BlowOffProcessedA,
	COM_GantryInPos 				:= IMD1_COM_IN.GantryA_Ready,
	COM_BlowOff_Pulse				=> IMD1_COM_OUT.BlowOffPulseA,
	COM_StartForming				=> IMD1_COM_OUT.StartFormingA, 
	COM_ErrSlotNotFree				=> IMD1_COM_OUT.ErrSlotANotFree,
);                                  

IMD1_GantryB(
	mxReset							:= mxReset,
	mxEmergency						:= mxEmergency,
	mxAutoMode						:= mxAutoMode,
	mrActModulo						:= mrActModPos,
	ProdPar							:= ProdParameters.BlowOff_Prod,
	COM_IMD_Stopped					:= IMD1_COM_IN.Stopped,
	COM_IMD_RTO						:= IMD1_COM_IN.RTO,
	COM_StartFormingReady			:= IMD1_COM_IN.FormingReadyB,
	COM_BlownOffProcessed			:= IMD1_COM_IN.BlowOffProcessedB,
	COM_GantryInPos 				:= IMD1_COM_IN.GantryB_Ready,
	COM_BlowOff_Pulse				=> IMD1_COM_OUT.BlowOffPulseB,
	COM_StartForming				=> IMD1_COM_OUT.StartFormingB, 
	COM_ErrSlotNotFree				=> IMD1_COM_OUT.ErrSlotBNotFree
); 


IMD2_GantryA(
	mxReset							:= mxReset,
	mxEmergency						:= mxEmergency,
	mxAutoMode						:= mxAutoMode,
	mrActModulo						:= mrActModPos,
	ProdPar							:= ProdParameters.BlowOff_Prod,
	COM_IMD_Stopped					:= IMD2_COM_IN.Stopped,
	COM_IMD_RTO						:= IMD2_COM_IN.RTO,
	COM_StartFormingReady			:= IMD2_COM_IN.FormingReadyA,
	COM_BlownOffProcessed			:= IMD2_COM_IN.BlowOffProcessedA,
	COM_GantryInPos 				:= IMD2_COM_IN.GantryA_Ready,
	COM_BlowOff_Pulse				=> IMD2_COM_OUT.BlowOffPulseA,
	COM_StartForming				=> IMD2_COM_OUT.StartFormingA, 
	COM_ErrSlotNotFree				=> IMD2_COM_OUT.ErrSlotANotFree
); 

IMD2_GantryB(
	mxReset							:= mxReset,
	mxEmergency						:= mxEmergency,
	mxAutoMode						:= mxAutoMode,
	mrActModulo						:= mrActModPos,
	ProdPar							:= ProdParameters.BlowOff_Prod,
	COM_IMD_Stopped					:= IMD2_COM_IN.Stopped,
	COM_IMD_RTO						:= IMD2_COM_IN.RTO,
	COM_StartFormingReady			:= IMD2_COM_IN.FormingReadyB,
	COM_BlownOffProcessed			:= IMD2_COM_IN.BlowOffProcessedB,
	COM_GantryInPos 				:= IMD2_COM_IN.GantryB_Ready,
	COM_BlowOff_Pulse				=> IMD2_COM_OUT.BlowOffPulseB,
	COM_StartForming				=> IMD2_COM_OUT.StartFormingB, 
	COM_ErrSlotNotFree				=> IMD2_COM_OUT.ErrSlotBNotFree
); 

Belt(
	mxEnable:= NOT mxEmergency, 
	mxInhibit:= FALSE, 
	mxAutoMode:= mxAutoMode, 
	mxReset:= mxReset, 
	mxEmergency:= mxEmergency, 
	mxSimulation:= , 
	mxFirstCycle:= , 
	mxResetCycle:= , 
	mxDisable_Positive:= FALSE, 
	mxDisable_Negative:= FALSE, 
	mxBlockHMI:= , 
	mrOverride:= 100.0, 
	mrVelocityManual:= MachParameters.VelocityManual, 
	SysParameters:= SysParameters.Belt,
	mxCycleBusy=> , 
	mxRunning=> , 
	Errors=> Errors.NCAxisError, 
	Error=> , 
	ErrorStop=> , 
	axStatus=> , 
	ActPosition=> , 
	ActVelocity=> , 
	axAxis=> );
END_ACTION

END_FUNCTION_BLOCK

// ---- Standard/NC_Axis/FB_NcAxis.TcPOU
FUNCTION_BLOCK FB_NcAxis
VAR CONSTANT

	sPosBiasStateTextDef: ARRAY[0..2] OF STRING:=	['State 0: Wait for Start',
										'State 1: Read Pos Bias, calculate new Pos Bias',
										'State 2: Write Pos Bias'];

	tPosBiasStateTimeouts: ARRAY[0..2] OF TIME:=  [T#10S, T#10S, T#10S];
	
END_VAR
VAR_INPUT
	mxEnable						: BOOL;
	mxInhibit						: BOOL :=TRUE;
	mxAutoMode						: BOOL;
	mxReset							: BOOL;
	mxFirstCycle					: BOOL;
	mxEmergency						: BOOL;
	mxSimulation					: BOOL;
	mxResetCycle					: BOOL;
	mxDisable_Positive				: BOOL; 
	mxDisable_Negative				: BOOL;
	mxBlockHMI						: BOOL:= FALSE;
	mrOverride						: LREAL;
	mrVelocityManual				: LREAL;
	mxResetPosBiasState				: BOOL;
	mxZeroCommand					: BOOL;
	mrHomePos						: LREAL;
END_VAR
VAR_IN_OUT
	SysParameters					: ST_NcAxis_SysPar;
END_VAR
VAR_OUTPUT
	mxCycleBusy						: BOOL;
	mxRunning						: BOOL;
	mxAxisIsMoving					: BOOL;
	///Errors
	Errors							: st_NcAxis_Errors;
	Error							: BOOL;
	ErrorStop						: BOOL;

	axStatus						:ST_AxisStatus;
	ActPosition						:LREAL;
	ActVelocity						:LREAL;

	axAxis							: AXIS_REF;

	mxPosBiasBusy					: BOOL;
	mxPosBiasHasError				: BOOL;
	SignalLightStatus					: BOOL;(* Needed in the HMI, for changing the color of the signal light *)	
END_VAR
VAR
	HmiStatus: UINT;
	HmiControl: UINT;
	HMI_ReadEncoder:BOOL;
	HMI_ReadmInc:LREAL;
	HMI_WriteEncoder:BOOL;
	HMI_WritemInc: LREAL;
	
	HMI_Forward				: BOOL;
	HMI_Backward			: BOOL;
	mxActivateAuto:BOOL;
	mxActivateManual:BOOL;
	mxActivated:BOOL;
	
	MCPower							: MC_Power;
	MCReset							: MC_Reset;
	MCJog							: MC_Jog;
	MCStop							: MC_Stop;
	MCHome							: MC_Home;
	MCMoveAbsolute					: ARRAY[0..1] OF MC_MoveAbsolute;
	mxMoveAbsNr						: INT;
	MCMoveVelocity					: ARRAY[0..1] OF MC_MoveVelocity;
	mxMoveVelocityNr				: INT;	
	MCReadParameter					: MC_ReadParameter;
	MCReadAxisError					: MC_ReadAxisError;
	MCWriteParameter				: MC_WriteParameter; 
 	MCSetPosition					: MC_SetPosition;
	MCReadStatus					: MC_ReadStatus;
	mcResetDrive					: FB_SoEReset_ByDriveRef;
	iDriveRef						AT %I* :ST_PLCDriveRef;
	
(*Drive parameters*)	
	mcBlendingMode					: MC_BufferMode;

	miState							: INT	:=0;
	miStopState						: INT	:=0;
	miOldstate						: INT	:=0;
	mxTransitionState				: BOOL	:= FALSE;
	sStateText						: STRING;	
	
 	exPosBiasTimeOut				: BOOL;		(* Timeout for the whole programcycle *)
	miPosBiasState					: INT	:=0;
	miPosBiasOldstate				: INT	:=0;
	mxPosBiasTransitionState		: BOOL	:= FALSE;
	sPosBiasStateText				: STRING;
	PosBiasTimeout					: TON;

(* Vars *)
	mxPosBiasTimeoutEnable			: BOOL;
	PosBiasTime						: REAL;

	mrStoredAxisPosition			: LREAL;
	mxPositionError					: BOOL;

	AdsReadPosBias					: ADSREAD;
	AdsWritePosBias					: ADSWRITE;

	PositionBiasRead 				: LREAL;
	
	(* Errors *)
	SR_DrivePower					: SR;
	SR_DriveJog						: SR;
	SR_DriveStatus					: SR;
	SR_DriveStop					: SR;
	SR_DriveReset					: SR;
	SR_Home							: SR;
	SR_Restart						: SR;
	SR_MotorError					: SR;
	SR_DriveAbsError				: SR;
	SR_DriveVelocity				: SR;
	SR_WriteParameter				: SR;
	SR_ReadParameter				: SR;
	SR_LagError						: SR;
 
	x: INT;
	
	mxCycleHasError					: BOOL;
	
(*Timers*)
	T_Power_On						: TON;
	T_Power_Off						: TOF;
	CycleTimeout					: TON;

(*Raising Edge detections*)
	RT_AutoManual					: R_TRIG;
	FT_AutoManual					: F_TRIG;
	RT_AutoManualHMI				: R_TRIG;
	CycleTimeOutUpFlank				: R_TRIG;
	PosBiasTimeOutUpFlank			: R_TRIG;

(* Vars *)
	mxCycleTimeoutEnable			: BOOL;
	CycleTime						: REAL;
	SR_CycleTimeOut					: SR;	
	mrPosition: LREAL;
	mrCheckPosition: LREAL;
	mxMoveForw: BOOL;
	mxSimulationDO	:INT:=0;	(*0= direct onposition, 1=seconds OnPosition, 2=not on position first and second*)
	ErrorIDMoveAbs1: UDINT;
	ErrorIDMoveAbs0: UDINT;

	T_Delay: TON;
	T_StandstillDelay: TON;
	miReadErrorID: DWORD;
	miReadAxisErrorID: DWORD;
END_VAR

Alarms();
WritePosBias();
HMI();
DriveActions();

ACTION Alarms:
SR_DrivePower(SET1:=MCPower.Error , RESET:=mxReset , Q1=> errors.exDrivePower);
SR_DriveJog(SET1:= MCJog.Error, RESET:=mxReset , Q1=> errors.exDriveJog);
SR_DriveStatus(SET1:= axAxis.Status.Error, RESET:=mxReset , Q1=> errors.exDriveStatus);
SR_DriveReset(SET1:= MCReset.Error, RESET:= mxReset, Q1=>errors.exDriveReset );
SR_DriveAbsError(SET1:=MCMoveAbsolute[0].Error OR MCMoveAbsolute[1].Error, RESET:= mxReset, Q1=>errors.exDriveAbsoluut );
SR_DriveStop(SET1:= MCStop.Error, RESET:= mxReset, Q1=>errors.exDriveStop );
SR_WriteParameter(SET1:= MCWriteParameter.Error, RESET:= mxReset, Q1=>errors.exWriteParameter );
SR_ReadParameter(SET1:= MCReadParameter.Error, RESET:= mxReset, Q1=>errors.exReadParameter );
SR_Home(SET1:= MCHome.Error, RESET:= mxReset, Q1=>errors.exHome );
SR_DriveVelocity(SET1:= MCMoveVelocity[0].Error OR MCMoveVelocity[0].Error, RESET:= mxReset, Q1=> Errors.exDriveVelocity);
SR_LagError(SET1:=(MCMoveAbsolute[0].ErrorID = 17744 AND MCMoveAbsolute[0].Error) OR 
						 (MCMoveAbsolute[1].ErrorID = 17744 AND MCMoveAbsolute[1].Error) OR
						 (MCJog.ErrorID = 17744 AND MCJog.Error) OR 
						 (MCMoveVelocity[0].ErrorID = 17744 AND MCMoveVelocity[0].Error) OR 
						 (MCMoveVelocity[1].ErrorID = 17744 AND MCMoveVelocity[1].Error) OR
						 axStatus.ErrorID = 17744
						 , RESET:= mxReset, Q1=>errors.exLagError );

ErrorStop:= errors.exLagError OR errors.exWriteParameter OR errors.exReadParameter OR 
	errors.exDriveStop OR errors.exDrivePower OR errors.exDriveJog  OR  errors.exDriveStatus OR 
	errors.exDriveReset OR Errors.exDriveAbsoluut OR Errors.exDriveVelocity OR errors.exHome;
END_ACTION

ACTION DriveActions:
(*read axis status*)
axAxis.ReadStatus();
axStatus:= axAxis.Status;
ActPosition:=axAxis.NcToPlc.ActPos;
ActVelocity:=axAxis.NcToPlc.ActVelo;
mxAxisIsMoving:= axAxis.Status.Moving;

	(*Power Axis*)
T_Power_On(IN:=(NOT mxInhibit), PT:= T#10MS);
T_Power_Off(IN:=T_Power_On.Q , PT:=T#5S , Q=> , ET=> );
(*power axis*)	
MCPower(
	Axis:= axAxis, 
	Enable:=NOT mxEmergency AND (T_Power_On.Q OR T_Power_Off.Q),  
	Enable_Positive:= NOT mxDisable_Positive , 
	Enable_Negative:= NOT mxDisable_Negative , 
	Override:=, 
	BufferMode:= , 
	Options:= , 
	Status=> , 
	Busy=> , 
	Active=> , 
	Error=> , 
	ErrorID=> );
	 
(*Drive run action manual*)
MCJog(
	Axis:= axAxis, 
	JogForward:= ,
	JogBackwards:= ,
	Mode:=MC_JOGMODE_CONTINOUS , 
	Position:= , 
	Velocity:= mrVelocityManual, 
	Acceleration:= , 
	Deceleration:= , 
	Jerk:= , 
	Done=> , 
	Busy=> , 
	Active=> , 
	CommandAborted=> , 
	Error=> , 
	ErrorID=> );
	MCJog.JogForward:=FALSE; 	
	MCJog.JogBackwards:=FALSE;

(*Drive Reset*)
MCReset(
	Axis:=axAxis , 
	Execute:=(mxReset AND (axAxis.Status.Error OR Error)), 
	Done=> , 
	Busy=> , 
	Error=> , 
	ErrorID=> );

	(*Reset*)
//DriveAxis.mcReset(Execute:= mxReset AND DriveAxis.mcStatus.Error, Axis:= axAxis);

(* Reset Drive Error *)
mcResetDrive.stDriveRef.sNetId:= F_CreateAmsNetId(iDriveRef.aNetId);
mcResetDrive.stDriveRef.nSlaveAddr:= iDriveRef.nSlaveAddr;
mcResetDrive.stDriveRef.nDriveNo:= iDriveRef.nDriveNo;


mcResetDrive(
	bExecute:= mxReset AND axAxis.Status.DriveDeviceError,
	tTimeout:= t#10s);
	
(*Move absolute fb 1*) 
	MCMoveAbsolute[0](
			Axis:= axAxis, 
			Execute:=, 
			Position:= , 
			Velocity:= , 
			Acceleration:= , 
			Deceleration:= , 
			Jerk:= , 
			BufferMode:= , 
			Options:= , 
			Done=> , 
			Busy=> , 
			Active=> , 
			CommandAborted=> , 
			Error=> , 
			ErrorID=> );
MCMoveAbsolute[0].Execute:=FALSE;
IF MCMoveAbsolute[0].ErrorID > 0 THEN ErrorIDMoveAbs0:=MCMoveAbsolute[0].ErrorID; END_IF;
(*Move absolute fb 2*)
	MCMoveAbsolute[1](
			Axis:= axAxis, 
			Execute:=, 
			Position:= , 
			Velocity:= , 
			Acceleration:= , 
			Deceleration:= , 
			Jerk:= , 
			BufferMode:=, 
			Options:= , 
			Done=> , 
			Busy=> , 
			Active=> , 
			CommandAborted=> , 
			Error=> , 
			ErrorID=>ErrorIDMoveAbs1 );
MCMoveAbsolute[1].Execute:=FALSE;
IF MCMoveAbsolute[1].ErrorID > 0 THEN ErrorIDMoveAbs0:=MCMoveAbsolute[1].ErrorID; END_IF;
(*Move velocity fb 1*)
MCMoveVelocity[0](
	Axis:=axAxis , 
	Execute:= , 
	Velocity:= , 
	Acceleration:= , 
	Deceleration:= , 
	Jerk:= , 
	Direction:= , 
	BufferMode:= , 
	Options:= , 
	InVelocity=> , 
	Busy=> , 
	Active=> , 
	CommandAborted=> , 
	Error=> , 
	ErrorID=> );
			
MCMoveVelocity[0].Execute:=FALSE;		
 (*Move velocity fb 2*)
MCMoveVelocity[1](
	Axis:=axAxis , 
	Execute:= , 
	Velocity:= , 
	Acceleration:= , 
	Deceleration:= , 
	Jerk:= , 
	Direction:= , 
	BufferMode:= , 
	Options:= , 
	InVelocity=> , 
	Busy=> , 
	Active=> , 
	CommandAborted=> , 
	Error=> , 
	ErrorID=> );
			
MCMoveVelocity[1].Execute:=FALSE;		

MCStop(
	Axis:=axAxis , 
	Execute:= , 
	Deceleration:= , 
	Jerk:= , 
	Options:= , 
	Done=> , 
	Busy=> , 
	Active=> , 
	CommandAborted=> , 
	Error=> , 
	ErrorID=> );
MCStop.Execute:=FALSE;

(*Homing*)
MCHome(
	Axis:=axAxis , 
	Execute:= , 
	Position:=  , 
	HomingMode:=  , 
	BufferMode:= , 
	Options:= , 
	bCalibrationCam:= , 
	Done=> , 
	Busy=> , 
	Active=> , 
	CommandAborted=> , 
	Error=> , 
	ErrorID=> );
MCHome.Execute:=FALSE;
	
(*Read a parameter*)
MCReadParameter(
	Axis:=axAxis , 
	Enable:= , 
	ParameterNumber:= , 
	ReadMode:=E_ReadMode.READMODE_CYCLIC , 
	Valid=> , 
	Busy=> , 
	Error=> , 
	ErrorID=> , 
	Value=> );
MCReadParameter.Enable:=FALSE;

(*Write a parameter*)	
MCWriteParameter(
	Axis:= axAxis, 
	Execute:= , 
	ParameterNumber:= , 
	Value:= , 
	Done=> , 
	Busy=> , 
	Error=> , 
	ErrorID=> );
MCWriteParameter.Execute:=FALSE;

MCSetPosition(
	Axis:= axAxis, 
	Execute:= , 
	Position:= , 
	Mode:=FALSE , 
	Options:= , 
	Done=> , 
	Busy=> , 
	Error=> , 
	ErrorID=> );
	MCSetPosition.Execute:=FALSE;	

MCReadAxisError(
	Axis:=axAxis , 
	Enable:=TRUE , 
	Valid=> , 
	Busy=> , 
	Error=> , 
	ErrorID=> miReadErrorID, 
	AxisErrorID=>miReadAxisErrorID );
	(*
MCReadStatus(
	Axis:= axAxis, 
	Enable:= , 
	Valid=> , 
	Busy=> , 
	Error=> , 
	ErrorID=> , 
	ErrorStop=> , 
	Disabled=> , 
	Stopping=> , 
	StandStill=> , 
	DiscreteMotion=> , 
	ContinuousMotion=> , 
	SynchronizedMotion=> , 
	Homing=> , 
	ConstantVelocity=> , 
	Accelerating=> , 
	Decelerating=> , 
	Status=> );*)
END_ACTION

ACTION HMI:
(*Read ax encoder parameter minc*)
IF HMI_ReadEncoder THEN
	HMI_ReadmInc :=	M_ReadParameter(MC_AxisParameter.AxisEncoderScalingFactor);
END_IF
(*Write ax encoder parameter*)
IF HMI_WriteEncoder THEN
	M_WriteParameter(miParameterNr:=MC_AxisParameter.AxisEncoderScalingFactor , miValue:= HMI_WritemInc );
END_IF

IF mxAutoMode THEN
	MCPower.Override:=mrOverride;
ELSE
	MCPower.Override:=mrOverride(*parameters.VelocityManual*);		
END_IF;

RT_AutoManual(CLK:= mxAutoMode);
FT_AutoManual(CLK:= mxAutoMode);

(*Set output*)
mxActivateAuto:= (mxEnable AND mxAutomode);
mxActivateManual := (mxEnable AND NOT mxAutoMode);

IF HMI_Forward AND axAxis.Status.Operational AND NOT SR_Restart.Q1 AND T_Power_On.Q AND NOT mxAutomode THEN
	MCJog.JogForward := TRUE ;
	MCJog.Velocity:= mrVelocityManual;
END_IF
IF HMI_Backward AND axAxis.Status.Operational AND NOT SR_Restart.Q1 AND T_Power_On.Q AND NOT mxAutoMode THEN
	MCJog.JogBackwards :=TRUE;
	MCJog.Velocity:= mrVelocityManual;
END_IF
END_ACTION

METHOD M_Home : BOOL;
VAR_INPUT
	mrHomePosition		: LREAL;
	MCMode				: MC_HomingMode;
END_VAR
McHome.Position:= mrHomePosition;
McHome.HomingMode:= MCMode;

McHome.Execute:= TRUE;


(* Return Value *)
M_Home:=MCHome.Done;
END_METHOD

METHOD M_MoveAbsolute : BOOL
VAR_INPUT
	Velocity				:LREAL;			
	Position				:LREAL;
END_VAR
(*compare for different setpoints, if so change fb mcMoveAbsolute*)
IF 	(MCMoveAbsolute[mxMoveAbsNr].Position <> Position) OR 
	(MCMoveAbsolute[mxMoveAbsNr].Velocity <> Velocity) THEN

	IF mxMoveAbsNr = 0 THEN
		mxMoveAbsNr :=1;
	ELSE
		mxMoveAbsNr :=0;
	END_IF
	
	(*Write parameters*)
	MCMoveAbsolute[mxMoveAbsNr].Position:=Position;
	MCMoveAbsolute[mxMoveAbsNr].Velocity:=Velocity;
(*	IF Velocity > 0.0 	THEN  MCMoveAbsolute[mxMoveAbsNr].Velocity:=Velocity; 		 ELSE MCMoveAbsolute[mxMoveAbsNr].Velocity:=parameters.VelocityAuto; 	END_IF*) 
END_IF

MCMoveAbsolute[mxMoveAbsNr].Execute:=TRUE;

(* Return value *)
M_MoveAbsolute:=MCMoveAbsolute[mxMoveAbsNr].Done;
END_METHOD

METHOD M_MoveVelocity : BOOL
VAR_INPUT
	Velocity			: LREAL;			
	Direction			: MC_Direction;
END_VAR
(*compare for different setpoints, if so change fb mcMoveVelocity*)
IF 	(MCMoveVelocity[mxMoveVelocityNr].Velocity <> Velocity) THEN

	IF mxMoveVelocityNr = 0 THEN
		mxMoveVelocityNr :=1;
	ELSE
		mxMoveVelocityNr :=0;
	END_IF

	(*Write parameters*)
	MCMoveVelocity[mxMoveVelocityNr].Velocity:=Velocity;
(*	IF Velocity > 0 	THEN MCMoveVelocity[mxMoveVelocityNr].Velocity:=Velocity; 			ELSE MCMoveVelocity[mxMoveVelocityNr].Velocity:=parameters.VelocityAuto; 		END_IF*)

END_IF

MCMoveVelocity[mxMoveVelocityNr].Execute:=TRUE;
MCMoveVelocity[mxMoveVelocityNr].Direction:=Direction;

(*Give return value*)
M_MoveVelocity:=MCMoveVelocity[mxMoveVelocityNr].Active;
END_METHOD

METHOD M_ReadParameter : LREAL
VAR_INPUT
		miParameterNr:INT;
END_VAR
MCReadParameter.ParameterNumber:=miParameterNr;
MCReadParameter.Enable:=TRUE;

M_ReadParameter:=MCReadParameter.Value;
END_METHOD

METHOD M_Reset : BOOL
VAR_INPUT
	
END_VAR

(* Return Value *)
M_Reset:= MCReset.Done;
END_METHOD

METHOD M_SetPosition : BOOL
VAR_INPUT
	NewPosition:LREAL;
END_VAR
MCSetPosition.Position:=NewPosition;
MCSetPosition.Execute:=TRUE;

M_SetPosition:=MCSetPosition.Done;
END_METHOD

METHOD M_Stop : BOOL
MCStop.Execute:=TRUE;

(* Return Value *)
M_Stop:= MCStop.Done;
END_METHOD

METHOD M_WriteParameter : BOOL
VAR_INPUT
	miParameterNr:INT;
	miValue:LREAL;
END_VAR
MCWriteParameter.ParameterNumber:=miParameterNr;
MCWriteParameter.Value:=miValue;
MCWriteParameter.Execute:=TRUE;

M_WriteParameter:=MCWriteParameter.Done;
END_METHOD

ACTION WritePosBias:
(*StateChange (Transition)  Signalgeneration*)
mxPosBiasTransitionState:=(miPosBiasState<>miPosBiasOldstate);
(*State text*)
sPosBiasStateText:=sPosBiasStateTextDef[miPosBiasState];
(*Timeout Watchdog for Statemachine*)
mxPosBiasTimeoutEnable:=NOT (miPosBiasState=0)  AND NOT mxReset;

PosBiasTimeout(IN:=mxPosBiasTimeoutEnable  , PT:=tPosBiasStateTimeouts[miPosBiasState] );
PosBiasTimeOutUpFlank(CLK:=PosBiasTimeout.Q );
miPosBiasOldstate:=miPosBiasState;

(*Set Errorbit when Raising edge of Timeout has been detected*)
IF PosBiasTimeOutUpFlank.Q THEN
	exPosBiasTimeOut:=TRUE; 			(* 1 Timeout for the whole programcycle *)
END_IF

(*Function to reset the Statemachine*)
IF mxResetPosBiasState THEN
	mxResetPosBiasState:=FALSE;
	miPosBiasState:=0;
	miPosBiasOldstate:=miPosBiasState;
	mxPosBiasTransitionState:=FALSE;

	AdsReadPosBias.READ:= FALSE;
	AdsWritePosBias.WRITE:= FALSE;

	mxZeroCommand:= FALSE;
	SignalLightStatus:= FALSE;
END_IF

AdsReadPosBias(
	NETID:= '',
	PORT:= 500,
	IDXGRP:= SysParameters.IDXGRP,
	IDXOFFS:= 16#7,
	LEN:= 8,
	DESTADDR:= ADR(PositionBiasRead),
	TMOUT:= T#1s);

AdsWritePosBias(
	NETID:= '',
	PORT:= 500,
	IDXGRP:= SysParameters.IDXGRP,
	IDXOFFS:= 16#7,
	LEN:= 8,
	SRCADDR:= ADR(SysParameters.PositionBias),
	TMOUT:= T#1s);

(*Definition State has Error*)
mxPosBiasHasError:=FALSE;

(*Cycle State's*)
CASE miPosBiasState OF
	(*Wait for Start *)
	0:
		(* Zero command from HMI *)
		IF mxZeroCommand THEN
			mxZeroCommand:= FALSE;
			SignalLightStatus:= FALSE;

			AdsReadPosBias.READ:= TRUE;
			miPosBiasState:= 1;
		END_IF

		(* PLC startup *)
		IF mxFirstCycle THEN
			SignalLightStatus:= FALSE;

			AdsWritePosBias.WRITE:= TRUE;
			miPosBiasState:= 2;
		END_IF

	(* Calculate new Position Bias with actual bias and act position *)
	1:
		IF NOT AdsReadPosBias.BUSY THEN
			AdsReadPosBias.READ:= FALSE;

			SysParameters.PositionBias:= mrHomePos - axAxis.NcToPlc.ActPos + PositionBiasRead;
			AdsWritePosBias.WRITE:= TRUE;

			miPosBiasState:= 2;
		END_IF

	(* Write new position bias *)
	2:
		IF NOT AdsWritePosBias.BUSY THEN
			AdsWritePosBias.WRITE:= FALSE;
			SignalLightStatus:= TRUE;

			miPosBiasState:= 0;
		END_IF
END_CASE

(*Set Busy bit FOR Statemachine*)
mxPosBiasBusy:=(miposBiasState<>0);
END_ACTION

END_FUNCTION_BLOCK

// ---- POUs/HMI.TcPOU
PROGRAM HMI
VAR_OUTPUT
	mxError		:BOOL; (*Error present*)
END_VAR

VAR

(*HMI Vars*)
	AlarmWord1 :DINT;	(* General *)
	AlarmWord2 :DINT;	(* General *)
	AlarmWord3 :DINT;	(* TopMold A *)
	AlarmWord4 :DINT;	(* TopMold A *)
	AlarmWord5 :DINT;	(* TopMold B *)
	AlarmWord6 :DINT;	(* TopMold B *)
	AlarmWord7 :DINT;	(* BottomMold A *)	
	AlarmWord8 :DINT;	(* BottomMold A *)
	AlarmWord9 :DINT;	(* BottomMold A *)
	AlarmWord10 :DINT;	(* BottomMold A *)
	AlarmWord11 :DINT;	(* BottomMold B *)
	AlarmWord12 :DINT;	(* BottomMold B *)
	AlarmWord13 :DINT;	(* BottomMold B *)
	AlarmWord14 :DINT;	(* BottomMold B *)
	AlarmWord15 :DINT;	(* TransferMold *)
	AlarmWord16 :DINT;	(* TransferMold *)
	AlarmWord17 :DINT;	(* ProductForming *)
	AlarmWord18 :DINT;	(* ProductForming *)
	AlarmWord19 :DINT;	(* ProductForming *)
	AlarmWord20 :DINT;	(* ProductForming *)


	sUserName	: STRING	:= 'NONE';
	miUserLevel	: INT		:= 0;

	mxReset		: BOOL;
	T_HmiReset	:TON;
	T_LogOut	: TON;

	mxAutoMode: BOOL;

END_VAR

Error();

T_HmiReset(IN:=mxReset,PT:=T#500MS);
IF T_HmiReset.Q THEN mxReset:=FALSE; END_IF

(********************************************************************
Automatically Logout after 10 minutes
********************************************************************)
T_LogOut(IN:=miUserLevel>0,PT:=t#10m);
IF T_LogOut.Q THEN
	miUserLevel := 0;
	sUserName := 'NONE';
END_IF

mxError:= AlarmWord1<>0 OR AlarmWord2<>0 OR AlarmWord3<>0 OR AlarmWord4<>0 OR AlarmWord5<>0 OR AlarmWord6<>0 OR
			AlarmWord7<>0 OR AlarmWord8<>0 OR AlarmWord9<>0 OR AlarmWord10<>0 OR AlarmWord11<>0 OR AlarmWord12<>0 OR
			AlarmWord13<>0 OR AlarmWord14<>0 OR AlarmWord15<>0 OR AlarmWord16<>0 OR AlarmWord17<>0 OR AlarmWord18<>0 OR
			AlarmWord19<>0 OR AlarmWord20<>0;

ACTION Error:
(*1*) AlarmWord1.0:= Main.Errors.exEmergency[1]; (* Zone error *)
(*2*) AlarmWord1.1:= Main.Errors.exEmergency[2];
(*3*) AlarmWord1.2:= Main.Errors.exEmergency[3];
(*4*) AlarmWord1.3:= Main.Errors.exEmergency[4];
(*5*) AlarmWord1.4:= Main.Errors.exEmergency[5];
(*6*) AlarmWord1.5:= Main.Errors.exEmergency[6];
(*7*) AlarmWord1.6:= Main.Errors.exEmergency[7];
(*8*) AlarmWord1.7:= FALSE;
(*9*) Alarmword1.8:= FALSE;
(*10*)Alarmword1.9:= FALSE;
(*11*)Alarmword1.10:=FALSE;
(*12*)Alarmword1.11:=FALSE;
(*13*)Alarmword1.12:=FALSE;
(*14*)Alarmword1.13:=FALSE;
(*15*)Alarmword1.14:=FALSE;
(*16*)Alarmword1.15:=FALSE;
(*17*)Alarmword1.16:=FALSE;
(*18*)Alarmword1.17:=FALSE;
(*19*)Alarmword1.18:=FALSE;
(*20*)Alarmword1.19:=FALSE;
(*21*)Alarmword1.20:=FALSE;
(*22*)Alarmword1.21:=FALSE;
(*23*)Alarmword1.22:=FALSE;
(*24*)Alarmword1.23:=FALSE;
(*25*)Alarmword1.24:=FALSE;
(*26*)Alarmword1.25:=FALSE;
(*27*)Alarmword1.26:=FALSE;
(*28*)Alarmword1.27:=FALSE;
(*29*)Alarmword1.28:=FALSE;
(*30*)Alarmword1.29:=FALSE;
(*31*)Alarmword1.30:=FALSE;
(*32*)Alarmword2.31:=FALSE;

(*33*)Alarmword2.0:= Main.Errors.ConveyorErrors.NCAxisError.exDriveAbsoluut;
(*34*)Alarmword2.1:= Main.Errors.ConveyorErrors.NCAxisError.exDriveJog;
(*35*)Alarmword2.2:= Main.Errors.ConveyorErrors.NCAxisError.exDrivePower;
(*36*)Alarmword2.3:= Main.Errors.ConveyorErrors.NCAxisError.exDriveReset;
(*37*)Alarmword2.4:= Main.Errors.ConveyorErrors.NCAxisError.exDriveStatus;
(*38*)Alarmword2.5:= Main.Errors.ConveyorErrors.NCAxisError.exDriveStop;
(*39*)Alarmword2.6:= Main.Errors.ConveyorErrors.NCAxisError.exDriveVelocity;
(*40*)Alarmword2.7:= Main.Errors.ConveyorErrors.NCAxisError.exHome;
(*41*)Alarmword2.8:= Main.Errors.ConveyorErrors.NCAxisError.exLagError;
(*42*)Alarmword2.9:= Main.Errors.ConveyorErrors.NCAxisError.exReadParameter;
(*43*)Alarmword2.10:=Main.Errors.ConveyorErrors.NCAxisError.exWriteParameter;
(*44*)Alarmword2.11:=FALSE;
(*45*)Alarmword2.12:=FALSE;
(*46*)Alarmword2.13:=FALSE;
(*47*)Alarmword2.14:=FALSE;
(*48*)Alarmword2.15:=FALSE;
(*49*)Alarmword2.16:=FALSE;
(*50*)Alarmword2.17:=FALSE;
(*51*)Alarmword2.18:=FALSE;
(*52*)Alarmword2.19:=FALSE;
(*53*)Alarmword2.20:=FALSE;
(*54*)Alarmword2.21:=FALSE;
(*55*)Alarmword2.22:=FALSE;
(*56*)Alarmword2.23:=FALSE;
(*57*)Alarmword2.24:=FALSE;
(*58*)Alarmword2.25:=FALSE;
(*59*)Alarmword2.26:=FALSE;
(*60*)Alarmword2.27:=FALSE;
(*61*)Alarmword2.28:=FALSE;
(*62*)Alarmword2.29:=FALSE;
(*63*)Alarmword2.30:=FALSE;
(*64*)Alarmword2.31:=FALSE;

(*65*)Alarmword3.0:=FALSE;
(*66*)Alarmword3.1:=FALSE;
(*67*)Alarmword3.2:=FALSE;
(*68*)Alarmword3.3:=FALSE;
(*69*)Alarmword3.4:=FALSE;
(*70*)Alarmword3.5:=FALSE;
(*71*)Alarmword3.6:=FALSE;
(*72*)Alarmword3.7:=FALSE;
(*73*)Alarmword3.8:=FALSE;
(*74*)Alarmword3.9:=FALSE;
(*75*)Alarmword3.10:=FALSE;
(*76*)Alarmword3.11:=FALSE;
(*77*)Alarmword3.12:=FALSE;
(*78*)Alarmword3.13:=FALSE;
(*79*)Alarmword3.14:=FALSE;
(*80*)Alarmword3.15:=FALSE;
(*81*)Alarmword3.16:=FALSE;
(*82*)Alarmword3.17:=FALSE;
(*83*)Alarmword3.18:=FALSE;
(*84*)Alarmword3.19:=FALSE;
(*85*)Alarmword3.20:=FALSE;
(*86*)Alarmword3.21:=FALSE;
(*87*)Alarmword3.22:=FALSE;
(*88*)Alarmword3.23:=FALSE;
(*89*)Alarmword3.24:=FALSE;
(*90*)Alarmword3.25:=FALSE;
(*91*)Alarmword3.26:=FALSE;
(*92*)Alarmword3.27:=FALSE;
(*93*)Alarmword3.28:=FALSE;
(*94*)Alarmword3.29:=FALSE;
(*95*)Alarmword3.30:=FALSE;
(*96*)Alarmword3.31:=FALSE;

(*97*)Alarmword4.0:=FALSE; 
(*98*)Alarmword4.1:=FALSE; 
(*99*)Alarmword4.2:=FALSE; 
(*100*)Alarmword4.3:=FALSE; 
(*101*)Alarmword4.4:=FALSE; 
(*102*)Alarmword4.5:=FALSE; 
(*103*)Alarmword4.6:=FALSE; 
(*104*)Alarmword4.7:=FALSE; 
(*105*)Alarmword4.8:=FALSE; 
(*106*)Alarmword4.9:=FALSE; 
(*107*)Alarmword4.10:=FALSE;
(*108*)Alarmword4.11:=FALSE;
(*109*)Alarmword4.12:=FALSE;
(*110*)Alarmword4.13:=FALSE;
(*111*)Alarmword4.14:=FALSE;
(*112*)Alarmword4.15:=FALSE;
(*113*)Alarmword4.16:=FALSE;
(*114*)Alarmword4.17:=FALSE;
(*115*)Alarmword4.18:=FALSE;
(*116*)Alarmword4.19:=FALSE;
(*117*)Alarmword4.20:=FALSE;
(*118*)Alarmword4.21:=FALSE;
(*119*)Alarmword4.22:=FALSE;
(*120*)Alarmword4.23:=FALSE;
(*121*)Alarmword4.24:=FALSE;
(*122*)Alarmword4.25:=FALSE;
(*123*)Alarmword4.26:=FALSE;
(*124*)Alarmword4.27:=FALSE;
(*125*)Alarmword4.28:=FALSE;
(*126*)Alarmword4.29:=FALSE;
(*127*)Alarmword4.30:=FALSE;
(*128*)Alarmword4.31:=FALSE;
END_ACTION

END_PROGRAM

// ---- POUs/SpeedControl/FB_BlowOff.TcPOU
FUNCTION_BLOCK FB_BlowOff
VAR CONSTANT
	sCycleStateTextDef: ARRAY[0..10]  OF STRING :=	
		['State 0: Wait for Start',
		'State 1: Calculate blowoff positions',
		'State 2: Blow off first sheet',
		'State 3: Blow off second sheet',
		'State 4: Blow off third sheet',
		'State 5: Blow off fourth sheet',
		'State 6: Start forming','7','8','9',
		'State 10: Slot Not Free Error'];
	
	tCycleStateTimeouts: ARRAY[0..10] OF TIME := 
		[T#10S,T#10S,T#60S,T#10S,T#10S,T#10S,T#10S,T#10S,T#10S,T#10S,
		T#10S];

END_VAR
VAR_INPUT
	mxResetCycleState				: BOOL;
	mxReset							: BOOL;	(*Reset Error*)
	mxEmergency						: BOOL;
	mxAutoMode						: BOOL; (* TRUE = Automode *)
	mxFirstCycle					: BOOL;
	
	mrActModulo						: LREAL;	//Modulo of main axis	
	mrModuloOffset					: LREAL;
	miSensorPitchClear				AT %I* : BOOL;
	ProdPar							: ST_BlowOffProdPar; 
	MachPar							: ST_BlowOffMachPar;
	
	COM_BlownOffProcessed			: ARRAY [1..4] OF BOOL;	
	COM_StartFormingReady			: BOOL;
	COM_IMD_RTO						: BOOL;
	COM_IMD_Stopped					: BOOL;
	COM_GantryInPos					: BOOL;
END_VAR
VAR_IN_OUT
	
END_VAR
VAR_OUTPUT
(*Errors*)
	Errors							: ST_BlowOffErrors;
	mxErrorStopinPos				: BOOL;		(* Error, stop in position. Only reset neccesary *)

(* State vars *)
	mxCycleBusy						: BOOL;
	
(* Vars *)	
	COM_BlowOff_Pulse				: ARRAY [1..4] OF BOOL;	
	COM_StartForming				: BOOL;
	COM_ErrSlotNotFree				: BOOL;
END_VAR
VAR
(* State vars *)
	miCycleState					: INT :=0;
	miCycleOldstate					: INT :=0;
	mxCycleTransitionState			: BOOL := FALSE;
	sCycleStateText					: STRING;
	exCycleTimeOut					: BOOL;		(* Timeout for the whole programcycle *)
	CycleTimeout					: TON;
	CycleTimeOutUpFlank				: R_TRIG;
	mxCycleTimeoutEnable			: BOOL;
	CycleTime						: REAL;
	mxCycleHasError					: BOOL;
	miStopState						: INT;
	mxStartCycle					: BOOL;
	mxStopCycle						: BOOL;
	mxStopDirect					: BOOL;
	
(* Internal vars for calculations *)
	BlowOff_Position				: ARRAY [1..4] OF LREAL;
	BlowOff_ResetTimer_Sheet1		: TON;
	BlowOff_ResetTimer_Sheet2		: TON;
	BlowOff_ResetTimer_Sheet3		: TON;
	BlowOff_ResetTimer_Sheet4		: TON;
	Forming_ResetTimer				: TON;
	ResetTime						: TIME;
	i								: DINT;
	mxWindowNotFree					: BOOL;
	mrModuloPosSensor				: LREAL;
	mrModuloPosSensorOffset			: LREAL;
	SensorFreeError_Time			: TIME;
	Timer_SensorFreeError			: TON;
	RT_SensorFree					: R_TRIG;
	RT_FormingReady					: R_TRIG;
	mxSensorOccupied				: BOOL;
	RT_SensorActivated				: R_TRIG;
	mrOldModulo						: LREAL;
	mrModuloDiffSensorActive		: LREAL;
	RT_NewCycle: R_TRIG;
	RT_IMD_Started: R_TRIG;
	RT_GantryAtPos: R_TRIG;
	mxNewCycleIMD: BOOL;
END_VAR

Error();
Cycle();

ACTION Cycle:
(*StateChange (Transition)  Signalgeneration*)
mxCycleTransitionState:=(miCycleState<>miCycleOldstate);
(*State text*)
sCycleStateText:=sCycleStateTextDef[miCycleState];
(*Timeout Watchdog for Statemachine*)
mxCycleTimeoutEnable:=NOT (miCycleState=0) AND NOT mxReset;

CycleTimeout(IN:=mxCycleTimeoutEnable, PT:=tCycleStateTimeouts[miCycleState] );
CycleTimeOutUpFlank(CLK:=CycleTimeout.Q );
miCycleOldstate:=miCycleState;

(*Set Errorbit when Raising edge of Timeout has been detected*)
IF CycleTimeOutUpFlank.Q THEN
	exCycleTimeOut:=TRUE; 			(* 1 Timeout for the whole programcycle *)
END_IF

(*Function to reset the Statemachine*)
IF mxResetCycleState THEN
	mxResetCycleState:= FALSE;
	miCycleState:=0;
	miCycleOldstate:=miCycleState;
	mxCycleTransitionState:=FALSE;

	mxStartCycle:= FALSE;
	mxStopCycle:= FALSE;
	mxStopDirect:= FALSE;
	COM_ErrSlotNotFree := FALSE;
END_IF

(*Blowoff times*)
	BlowOff_ResetTimer_Sheet1(IN:=COM_BlowOff_Pulse[1], PT:=ResetTime);
	IF BlowOff_ResetTimer_Sheet1.Q THEN
		COM_BlowOff_Pulse[1] := FALSE;
	END_IF
	
	BlowOff_ResetTimer_Sheet2(IN:=COM_BlowOff_Pulse[2], PT:=ResetTime);
	IF BlowOff_ResetTimer_Sheet2.Q THEN
		COM_BlowOff_Pulse[2] := FALSE;
	END_IF
	
	BlowOff_ResetTimer_Sheet3(IN:=COM_BlowOff_Pulse[3], PT:=ResetTime);
	IF BlowOff_ResetTimer_Sheet3.Q THEN
		COM_BlowOff_Pulse[3] := FALSE;
	END_IF
	
	BlowOff_ResetTimer_Sheet4(IN:=COM_BlowOff_Pulse[4], PT:=ResetTime);
	IF BlowOff_ResetTimer_Sheet4.Q THEN
		COM_BlowOff_Pulse[4] := FALSE;
	END_IF	

(*Forming signal to IMD*)
	RT_IMD_Started(CLK:=COM_IMD_RTO AND NOT COM_IMD_Stopped);
	RT_GantryAtPos(CLK:=COM_GantryInPos);
	IF RT_IMD_Started.Q THEN
		mxNewCycleIMD := TRUE;
	END_IF
	IF RT_GantryAtPos.Q THEN
		mxNewCycleIMD := FALSE;
	END_IF

	RT_FormingReady(CLK:=COM_StartFormingReady);
	RT_NewCycle(CLK:= miCycleState = 3);
	IF RT_FormingReady.Q OR RT_NewCycle.Q OR NOT COM_IMD_RTO THEN
		COM_StartForming := FALSE;
	END_IF
		
	
	
(*Definition State has Error*)
mxCycleHasError:=FALSE;

(*Modulo position Sensor Free detection*)
	IF (ProdPar.NrOfSheets <> 0) AND (ProdPar.SheetSize <> 0 ) THEN
		mrModuloPosSensorOffset := ProdPar.ModuloOffsetSensorFree + (ProdPar.SheetSize/2) + (((DINT_TO_REAL(ProdPar.NrOfSheets)/2) - 0.5) * ProdPar.PitchGantry);
	ELSE
		mrModuloPosSensorOffset := ProdPar.ModuloOffsetSensorFree;
	END_IF
	
	IF (mrModuloOffset - mrModuloPosSensorOffset) < 0 THEN
		mrModuloPosSensor := ProdPar.Modulo + (mrModuloOffset - mrModuloPosSensorOffset);	
	ELSE
		mrModuloPosSensor := mrModuloOffset - mrModuloPosSensorOffset;
	END_IF

	IF mxCycleBusy THEN
		IF (mrModuloOffset - mrModuloPosSensorOffset) < 0 THEN
			IF (mrActModulo >= mrModuloPosSensor) OR (mrActModulo <= (mrModuloOffset - mrModuloPosSensorOffset + (ProdPar.Modulo/4))) THEN						
				mxSensorOccupied := miSensorPitchClear;
				//Timer_SensorFreeError.IN:= miSensorPitchClear;
			ELSE 
				mxSensorOccupied := FALSE;
			END_IF
		ELSE
			IF (mrActModulo >= mrModuloPosSensor) AND (mrActModulo <= (mrModuloOffset - mrModuloPosSensorOffset + (ProdPar.Modulo/4))) THEN		
				mxSensorOccupied := miSensorPitchClear;
				//Timer_SensorFreeError.IN:= miSensorPitchClear;
			ELSE
				mxSensorOccupied := FALSE;
			END_IF
		END_IF
	ELSE
		//Timer_SensorFreeError.IN:= FALSE;
		mxSensorOccupied := FALSE;
	END_IF
	
	RT_SensorActivated(CLK:= mxSensorOccupied);
	
	IF RT_SensorActivated.Q THEN
		mrOldModulo := mrActModulo;
	END_IF
	
	IF mxSensorOccupied THEN
		IF mrActModulo < mrOldModulo THEN
			mrModuloDiffSensorActive := (ProdPar.Modulo - mrOldModulo) + mrActModulo;	
		ELSE
			mrModuloDiffSensorActive := mrActModulo - mrOldModulo;	
		END_IF
		IF mrModuloDiffSensorActive >= ProdPar.ModuloDetectionSensorFree THEN
			COM_ErrSlotNotFree := TRUE;
		END_IF 
	ELSE
		mrModuloDiffSensorActive := 0;
	END_IF
	
	(*Timer_SensorFreeError();
	IF Timer_SensorFreeError.Q THEN
		Timer_SensorFreeError.IN:= FALSE;
		COM_ErrSlotNotFree := TRUE;
	END_IF*)	

(*Cycle State's*)
CASE miCycleState OF
	0:	//Wait for start Cycle
		IF mxStartCycle THEN
			mxStartCycle:= FALSE;

			miCycleState:= 1;
			COM_ErrSlotNotFree := FALSE;
		END_IF	

	1: //Blow off first sheet
		IF mxStopDirect THEN
			mxStopDirect:= FALSE;
			
			miCycleState:= 25;
		ELSIF mxStopCycle THEN
			mxStopCycle:= FALSE;

			miStopState:= miCycleState;
			miCycleState:= 20;
		ELSE
			i := 1;
			WHILE i <= ProdPar.NrOfSheets DO  
				IF i > 1 THEN
					//Calculate blowoff positions:
					BlowOff_Position[i] := ((((ProdPar.Modulo/4)/ProdPar.NrOfSheets) - (ProdPar.PitchGantry + 1)) * (i - 1)) +  mrModuloOffset;
				ELSE
					BlowOff_Position[i] := mrModuloOffset;
				END_IF
			
				i := i + 1;
			END_WHILE

			miCycleState := 2;
		END_IF

	2:	//Blowoff first sheet
		IF mxStopDirect THEN
			mxStopDirect:= FALSE;
			
			miCycleState:= 25;
		ELSIF mxStopCycle THEN
			mxStopCycle:= FALSE;

			miStopState:= miCycleState;
			miCycleState:= 20;
		ELSIF COM_ErrSlotNotFree THEN
			miCycleState := 10;
		ELSE 
			//Create blowoff pulse
			IF mrActModulo >= BlowOff_Position[1] AND mrActModulo <  (BlowOff_Position[1]+10) THEN
				COM_BlowOff_Pulse[3] := TRUE;		//MZE 20190327 	COM_BlowOff_Pulse[1] for HLU and COM_BlowOff_Pulse[3] for LoodsLanghout  		
				miCycleState := 3; 
			END_IF
		END_IF
		
	3:	//Blowoff Second sheet
		IF mxStopDirect THEN
			mxStopDirect:= FALSE;
			
			miCycleState:= 25;
		ELSIF mxStopCycle THEN
			mxStopCycle:= FALSE;

			miStopState:= miCycleState;
			miCycleState:= 20;
		ELSIF COM_ErrSlotNotFree THEN
			miCycleState := 10;
		ELSE
			IF ProdPar.NrOfSheets >= 2 THEN 
				//Create blowoff pulse
				IF mrActModulo >= BlowOff_Position[2] THEN 
					COM_BlowOff_Pulse[2] := TRUE;	
					miCycleState := 4;
				END_IF
			ELSE
				miCycleState := 6; //Go to Start Forming;
			END_IF
		END_IF
	
	4:	//Blowoff Third sheet
		IF mxStopDirect THEN
			mxStopDirect:= FALSE;
			
			miCycleState:= 25;
		ELSIF mxStopCycle THEN
			mxStopCycle:= FALSE;

			miStopState:= miCycleState;
			miCycleState:= 20;
		ELSIF COM_ErrSlotNotFree THEN
			miCycleState := 10;
		ELSE
			IF ProdPar.NrOfSheets >= 3 THEN 
				//Create blowoff pulse
				IF mrActModulo >= BlowOff_Position[3] THEN	
					COM_BlowOff_Pulse[1] := TRUE;			//MZE 20190327 	COM_BlowOff_Pulse[3] for HLU and COM_BlowOff_Pulse[1] for LoodsLanghout
					miCycleState := 5;
				END_IF
			ELSE
				miCycleState := 6; //Go to Start Forming;
			END_IF
		END_IF
		
	5:	//Blowoff Fourth sheet
		IF mxStopDirect THEN
			mxStopDirect:= FALSE;
			
			miCycleState:= 25;
		ELSIF mxStopCycle THEN
			mxStopCycle:= FALSE;

			miStopState:= miCycleState;
			miCycleState:= 20;
		ELSIF COM_ErrSlotNotFree THEN
			miCycleState := 10;
		ELSE
			IF ProdPar.NrOfSheets >= 4 THEN 
				//Create blowoff pulse
				IF mrActModulo >= BlowOff_Position[4] THEN
					COM_BlowOff_Pulse[4] := TRUE;
					miCycleState := 6;
				END_IF
			ELSE
				miCycleState := 6; //Go to Start Forming;
			END_IF
		END_IF
		
	6:	//Start Forming
		IF mxStopDirect THEN
			mxStopDirect:= FALSE;
			
			miCycleState:= 25;
		ELSIF mxStopCycle THEN
			mxStopCycle:= FALSE;

			miStopState:= miCycleState;
			miCycleState:= 20;
		ELSE
			IF COM_IMD_RTO AND NOT COM_IMD_Stopped THEN
				COM_StartForming := TRUE;
			END_IF
			miCycleState := 2;
		END_IF
		
	10:	//Error slot not free
		IF mxStopDirect THEN
			mxStopDirect:= FALSE;
			
			miCycleState:= 25;
		ELSIF mxStopCycle THEN
			mxStopCycle:= FALSE;

			miStopState:= miCycleState;
			miCycleState:= 20;
		ELSE 
			IF mrActModulo >= (mrModuloOffset + (ProdPar.Modulo/4) - 10) THEN 
				COM_ErrSlotNotFree := FALSE; 
				miCycleState := 2;
			END_IF
		END_IF
		
	(* Stop Cycle, stop belt after x mm*)
	20:
		IF mxStopDirect THEN
			mxStopDirect:= FALSE;
			
			miCycleState:= 25;
		ELSE 
			mxStopCycle:= FALSE;
			miCycleState:= 21;
		END_IF

	(* stopped, wait for restart*)	
	21:
		IF mxStopDirect THEN
			mxStopDirect:= FALSE;
	
			miCycleState:= 25;
		ELSIF mxStartCycle THEN
			mxStartCycle := FALSE;
			miCycleState := miStopState;
		END_IF	
		
		
	(* Stop Direct *)
	25:
		mxStartCycle:= FALSE;
		mxStopCycle:= FALSE;
		mxStopDirect:= FALSE;
		
		
		miCycleState:= 0;
END_CASE

mxCycleBusy:= miCycleState<>0 AND miCycleState <>21 ;
END_ACTION

ACTION Error:


(*************************************************************************************************)
mxErrorStopinPos:= FALSE;
END_ACTION

METHOD M_StartCycle

IF NOT mxCycleBusy THEN
	mxStartCycle:= TRUE;	
END_IF
END_METHOD

METHOD M_StopCycle

IF mxCycleBusy THEN 
	mxStopCycle:= TRUE; 
END_IF
END_METHOD

METHOD M_StopDirect

IF mxCycleBusy THEN
	mxStopDirect:= TRUE;	
END_IF
END_METHOD

END_FUNCTION_BLOCK

// ---- Standard/FB_Blink.TcPOU
FUNCTION_BLOCK FB_Blink
VAR_INPUT
END_VAR
VAR_OUTPUT
	Fast:BOOL;
	Normal:BOOL;
	Slow:BOOL;
END_VAR
VAR
	TFast:TON;
	TNormal:TON;
	TSlow:TON;

END_VAR

TFast(IN:=NOT TFast.Q , PT:=T#0.1S);
TNormal(IN:=NOT TNormal.Q , PT:=T#0.2S);
TSlow(IN:=NOT TSlow.Q , PT:=T#0.3S);

IF TFast.Q THEN
	(*Toggle bit*)
	Fast:=NOT Fast;
END_IF

IF TNormal.Q THEN
	(*Toggle bit*)
	Normal:=NOT Normal;
END_IF

IF TSlow.Q THEN
	(*Toggle bit*)
	Slow:=NOT Slow;
END_IF

END_FUNCTION_BLOCK

// ---- Standard/FB_EthercatDiag.TcPOU
FUNCTION_BLOCK FB_EtherCATDiag
VAR_INPUT
(* EtherCAT *)
	SlaveCount 		:UINT;		(* Actual count of EtherCAT slaves received *)
	CfgSlaveCount	:UINT;		(* Count of configured EtherCAT slaves *)

	DevState 		:UINT;		(* EtherCAT State:
									0x0001 = Link error
									0x0002 = I/O locked after link error (I/O reset required)
									0x0004 = Link error (redundancy adapter)
									0x0008 = Missing one frame (redundancy mode)
									0x0010 = Out of send resources (I/O reset required)
									0x0020 = Watchdog triggered
									0x0040 = Ethernet driver (miniport) not found
									0x0080 = I/O reset active
									0x0100 = At least one device in 'INIT' state
									0x0200 = At least one device in 'PRE-OP' state
									0x0400 = At least one device in 'SAFE-OP' state
									0x0800 = At least one device indicates an error state
									0x1000 = DC not in sync
								 *)
END_VAR

VAR_OUTPUT
(* Alarms*)
	EtherCATLinkError			: BOOL;		(* EtherCAT error, link error *)
	EtherCATSlaveMissing		: BOOL;		(* EtherCAT error, at least one device not connected *)
	EtherCATOPmode				: BOOL;		(* EtherCAT error, at leat one device not in 'OP'-mode *)
	EtherCATResetNeeded			: BOOL;		(* EtherCAT error, I/O reset required *)
END_VAR

VAR
	Fx: WORD;

	bInit						: BOOL;		(* At least one device in 'INIT' state *)
	bPreOP						: BOOL;		(* At least one device in 'PRE-OP' state *)
	bSafeOP						: BOOL;		(* At least one device in 'SAFE-OP' state *)
	bError						: BOOL;		(* At least one device indicates an error state *)
	bIOLocked					: BOOL;		(* I/O locked after link error (I/O reset required) *)
	bNoResources				: BOOL;		(* Out of send resources (I/O reset required) *)
END_VAR

(*----------------------------------------------------------------------------------------------------------------*)
(* Slave missing form EtherCAT bus *)
(* Alarm message: EtherCAT error, at least one device not connected *)
IF SlaveCount <> CfgSlaveCount
THEN
	EtherCATSlaveMissing	:= TRUE;
ELSE
	EtherCATSlaveMissing	:= FALSE;
END_IF


(*----------------------------------------------------------------------------------------------------------------*)
(* EtherCAT device link error *)
Fx := UINT_TO_WORD(DevState) AND 16#0001;

IF Fx = 16#0001
THEN
	EtherCATLinkError := TRUE;
ELSE
	EtherCATLinkError := FALSE;
END_IF


(*----------------------------------------------------------------------------------------------------------------*)
(* EtherCAT device not in 'OP'-mode *)
(* Check devices for INIT-state *)
Fx	:= UINT_TO_WORD( DevState ) AND 16#0100;

IF Fx = 16#0100
THEN
	bInit		:= TRUE;
ELSE
	bInit 		:= FALSE;
END_IF

(* Check devices for PREOP-state *)
Fx := UINT_TO_WORD( DevState ) AND 16#0200;

IF Fx = 16#0200
THEN
	bPreOP		:= TRUE;
ELSE
	bPreOP 		:= FALSE;
END_IF

(* Check devices for SAFEEOP-state *)
Fx := UINT_TO_WORD( DevState ) AND 16#0400;

IF Fx = 16#0400
THEN
	bSafeOP		:= TRUE;
ELSE
	bSafeOP 	:= FALSE;
END_IF

(* Check devices for error-state *)
Fx := UINT_TO_WORD( DevState ) AND 16#0800;

IF Fx = 16#0800
THEN
	bError		:= TRUE;
ELSE
	bError 		:= FALSE;
END_IF

(* At least one device not in OP-mode *)
EtherCATOPmode	:=			bInit
						OR	bPreOP
						OR	bSafeOP
						OR	bError;


(*----------------------------------------------------------------------------------------------------------------*)
(* EtherCAT I/O reset needed *)
(* Check for any I/O lock *)
Fx := UINT_TO_WORD( DevState ) AND 16#0002;

IF Fx = 16#0002
THEN
	bIOLocked		:= TRUE;
ELSE
	bIOLocked 		:= FALSE;
END_IF

(* Check for out of send resources *)
Fx := UINT_TO_WORD( DevState ) AND 16#0010;

IF Fx = 16#0010
THEN
	bNoResources		:= TRUE;
ELSE
	bNoResources 		:= FALSE;
END_IF

(* EtherCAT error, I/O reset required *)
EtherCATResetNeeded	:=			bIOLocked
							OR	bNoResources;

END_FUNCTION_BLOCK

// ---- Standard/Motor/FB_Motor.TcPOU
FUNCTION_BLOCK FB_Motor
VAR_INPUT
	mxReset							: BOOL;
	mxEmergency						: BOOL;
	mxAutoMode						: BOOL;
	mxDisableManualAutoTrigger		: BOOL := FALSE; // If this bit is enabled, the outputs status is not changed when change from/to automode happens
END_VAR
VAR_OUTPUT
(*Errors*)
	Errors							: ST_MotorErrors;
	mxErrorInit						: BOOL;		(* Error, stop immediately. Initialisation neccesary *)
	mxErrorStopinPos				: BOOL;		(* Error, stop in position. Only reset neccesary *)

(* State vars *)
	mxCycleBusy						: BOOL;
	mxInitBusy						: BOOL;
	
(* Vars *)
	mxInitialized					: BOOL;
	IsRunning						: BOOL;
	
END_VAR
VAR
	ixThermal						AT %I* : BOOL;
	ixRunning						AT %I* : BOOL;
	ixMaintenance					AT %I* : BOOL;
	Q								AT %Q* : BOOL;
	
	Hmi_On							: BOOL;
	RT_AutoMode						: R_TRIG;
	SR_ErrorThermal					: SR;
	SR_ErrorMaintenance				: SR;
	Ixtest: BOOL;
END_VAR

Error();

(* Reset hmi when switched to automode*)
RT_AutoMode(CLK:= mxAutoMode);

// if manual mode becomes active, the manualmode (hmi) is over written by its current state.
// this ensures that the motor keeps running when it was running and is switched to manual. 
IF RT_AutoMode.Q AND NOT mxDisableManualAutoTrigger THEN Hmi_On:= Q; END_IF	

(* Manual control *)
//IF NOT mxAutoMode THEN Q:= Hmi_On; END_IF

// Is running becomes high when signal becomes low.
IsRunning:= NOT ixRunning;

ACTION Error:
SR_ErrorThermal(SET1:= NOT ixThermal, RESET:= mxReset, Q1=> Errors.Thermal);
SR_ErrorMaintenance(SET1:= NOT ixMaintenance, RESET:= mxReset, Q1=> Errors.Maintenance);

(******************************************************************************************************)
mxErrorStopinPos:= FALSE;
mxErrorInit:= Errors.Thermal OR Errors.Maintenance;
END_ACTION

METHOD M_Init

Q:= FALSE;
END_METHOD

METHOD M_Start : BOOL
VAR_INPUT
END_VAR
Q:=TRUE;

(* Return Value *)
M_Start:= Q;
END_METHOD

METHOD M_Stop : BOOL
VAR_INPUT
END_VAR
Q:= FALSE;

(* Return Value *)
M_Stop:= NOT Q;
END_METHOD

END_FUNCTION_BLOCK

// ---- Standard/Motor/FB_MotorSS.TcPOU
FUNCTION_BLOCK FB_MotorSS
VAR_INPUT
	mxReset							: BOOL;
	mxEmergency						: BOOL;
	mxAutoMode						: BOOL;
	mxDisableManualAutoTrigger		: BOOL := FALSE; // If this bit is enabled, the outputs status is not changed when change from/to automode happens
END_VAR
VAR_OUTPUT
(*Errors*)
	Errors							: ST_MotorSSErrors;
	mxErrorInit						: BOOL;		(* Error, stop immediately. Initialisation neccesary *)
	mxErrorStopinPos				: BOOL;		(* Error, stop in position. Only reset neccesary *)

(* State vars *)
	mxCycleBusy						: BOOL;
	mxInitBusy						: BOOL;
	
(* Vars *)
	mxInitialized					: BOOL;
	IsRunning						: BOOL;
	
END_VAR
VAR
	ixSSFailure						AT %I* : BOOL;
	ixMaintenance					AT %I* : BOOL;
	ixIsRunning						AT %I* : BOOL;
	Q								AT %Q* : BOOL;
	
	Hmi_On							: BOOL;
	RT_AutoMode						: R_TRIG;
	SR_ErrorMaintenance				: SR;
	SR_ErrorSS: SR;
	mxTest: BOOL;
END_VAR

Error();

(* Reset hmi when switched to automode*)
RT_AutoMode(CLK:= mxAutoMode);

// if manual mode becomes active, the manualmode (hmi) is over written by its current state.
// this ensures that the motor keeps running when it was running and is switched to manual. 
IF RT_AutoMode.Q AND NOT mxDisableManualAutoTrigger THEN Hmi_On:= Q; END_IF	

(* Manual control *)
//IF NOT mxAutoMode THEN Q:= Hmi_On; END_IF

IsRunning:= ixIsRunning;

ACTION Error:
SR_ErrorSS(SET1:= NOT ixSSFailure, RESET:= mxReset, Q1=> Errors.SofstarterFailure);
SR_ErrorMaintenance(SET1:= NOT ixMaintenance, RESET:= mxReset, Q1=> Errors.Maintenance);

(******************************************************************************************************)
mxErrorStopinPos:= FALSE;
mxErrorInit:= Errors.SofstarterFailure OR Errors.Maintenance;
END_ACTION

METHOD M_Init

Q:= FALSE;
END_METHOD

METHOD M_Start : BOOL
VAR_INPUT
END_VAR
Q:=TRUE;

(* Return Value *)
M_Start:= Q;
END_METHOD

METHOD M_Stop : BOOL
VAR_INPUT
END_VAR
Q:= FALSE;

(* Return Value *)
M_Stop:= NOT Q;
END_METHOD

END_FUNCTION_BLOCK
